(* CODESYS project tcunit.library
   Company: www.tcunit.org
   DefaultNamespace: TcUnit
   Version: 1.0.0.0
   Placeholder: TcUnit
   Author: Jakob Sagatowski and contributors
   Description: TwinCAT unit testing framework.
      Documentation and examples are available at www.tcunit.org
   Title: TcUnit

Project tree, tasks and I/O mapping:
  libraries: Base Interfaces, * (System); SysFile, * (System); Tc2_Standard, * (Beckhoff Automation GmbH); Tc2_System, * (Beckhoff Automation GmbH); Tc2_Utilities, * (Beckhoff Automation GmbH)
  DUTs/
    data type E_XmlError
    data type ST_ADSLogStringMessage
    data type ST_AssertArrayResult
    data type ST_AssertArrayResultInstances
    data type ST_AssertResult
    data type ST_AssertResultInstances
    data type U_ExpectedOrActual
  GVLs/
    global variables GVL_Param_TcUnit
    global variables GVL_Param_XmlControl
    global variables GVL_TcUnit
  ITFs/
    interface I_AssertMessageFormatter: LogAssertFailure
    interface I_TestResultFormatter: Format
  POUs/
    Functions/
      WRITE_PROTECTED_/
        function WRITE_PROTECTED_BOOL [ST]
        function WRITE_PROTECTED_BYTE [ST]
        function WRITE_PROTECTED_DATE [ST]
        function WRITE_PROTECTED_DATE_AND_TIME [ST]
        function WRITE_PROTECTED_DINT [ST]
        function WRITE_PROTECTED_DWORD [ST]
        function WRITE_PROTECTED_INT [ST]
        function WRITE_PROTECTED_LREAL [ST]
        function WRITE_PROTECTED_REAL [ST]
        function WRITE_PROTECTED_SINT [ST]
        function WRITE_PROTECTED_STRING [ST]
        function WRITE_PROTECTED_TIME [ST]
        function WRITE_PROTECTED_TIME_OF_DAY [ST]
        function WRITE_PROTECTED_UDINT [ST]
        function WRITE_PROTECTED_UINT [ST]
        function WRITE_PROTECTED_USINT [ST]
        function WRITE_PROTECTED_WORD [ST]
      function F_AnyToUnionValue [ST]
      function F_AnyTypeClassToString [ST]
      function F_IsAnyEqualToUnionValue [ST]
      function F_RemoveInstancePathAndProjectNameFromTestInstancePath [ST]
      function IS_TEST_FINISHED [ST]
      function RUN [ST]
      function TEST [ST]
      function TEST_FINISHED [ST]
      function TEST_FINISHED_NAMED [ST]
    function block FB_AdjustAssertFailureMessageToMax252CharLength [ST]
    function block FB_ADSAssertMessageFormatter [ST]: LogAssertFailure
    function block FB_ADSLogStringMessageFifoQueue [ST]: GetLog, GetLogCount, WriteLog
    function block FB_ADSTestResultFormatter [ST]: Format
    function block FB_AnyComparator [ST]
    function block FB_AssertArrayResultStatic [ST]: AddAssertArrayResult, CopyDetectionCountAndResetDetectionCountInThisCycle, CreateAssertResultInstance, GetDetectionCount, GetDetectionCountThisCycle, IncreaseDetectionCountThisCycleByOne, ReportResult
    function block FB_AssertResultStatic [ST]: AddAssertResult, CopyDetectionCountAndResetDetectionCountInThisCycle, CreateAssertResultInstance, GetDetectionCount, GetDetectionCountThisCycle, IncreaseDetectionCountThisCycleByOne, ReportResult
    function block FB_FileControl [ST]: Close, Open, Read, Save
    function block FB_StringBuffer [ST]: Append, BufferSize, Copy, CutOff, Find, FindBack, Length, Set
    function block FB_TcUnitRunner [ST]: AbortRunningTestSuiteTests, RunTestSuiteTests
    function block FB_Test [ST]: GetName, IsFailed, IsFinished, SetFailed, SetFinished, SetName
    function block FB_TestSuite [ST]: AddTest, AddTestNameToInstancePath, AreAllTestsFinished, AssertArray2dEquals_LREAL, AssertArray2dEquals_REAL, AssertArray3dEquals_LREAL, AssertArray3dEquals_REAL, AssertArrayEquals_BOOL, AssertArrayEquals_BYTE, AssertArrayEquals_DINT, AssertArrayEquals_DWORD, AssertArrayEquals_INT, AssertArrayEquals_LINT, AssertArrayEquals_LREAL, AssertArrayEquals_LWORD, AssertArrayEquals_REAL, AssertArrayEquals_SINT, AssertArrayEquals_UDINT, AssertArrayEquals_UINT, AssertArrayEquals_ULINT, AssertArrayEquals_USINT, AssertArrayEquals_WORD, AssertEquals, AssertEquals_BOOL, AssertEquals_BYTE, AssertEquals_DATE, AssertEquals_DATE_AND_TIME, AssertEquals_DINT, AssertEquals_DWORD, AssertEquals_INT, AssertEquals_LINT, AssertEquals_LREAL, AssertEquals_LTIME, AssertEquals_LWORD, AssertEquals_REAL, AssertEquals_SINT, AssertEquals_STRING, AssertEquals_TIME, AssertEquals_TIME_OF_DAY, AssertEquals_UDINT, AssertEquals_UINT, AssertEquals_ULINT, AssertEquals_USINT, AssertEquals_WORD, AssertFalse, AssertTrue, FB_init, FindTestSuiteInstancePath, GetInstancePath, GetNumberOfFailedTests, GetNumberOfSuccessfulTests, GetNumberOfTests, SetTestFailed, SetTestFinished
    function block FB_XmlControl [ST]: ClearBuffer, CloseTag, Length, NewComment, NewParameter, NewTag, NewTagData, NextParameter, NextTag, SetBuffer, ToStartBuffer, WriteDocumentHeader
  Version/
    global variables Global_Version
*)

// DUTs/E_XmlError
{attribute 'qualified_only'}
{attribute 'strict'}
TYPE E_XmlError :
(
    Ok := 0,
    ErrorMaxBufferLen := 1,
    ErrorStringLen := 2,
    Error := 3
) BYTE;
END_TYPE

// DUTs/ST_ADSLogStringMessage
{attribute 'pack_mode' := '1'}
TYPE ST_ADSLogStringMessage :
STRUCT
    MsgFmtStr : Tc2_System.T_MaxString;
    StrArg : Tc2_System.T_MaxString;
END_STRUCT
END_TYPE

// DUTs/ST_AssertArrayResult
TYPE ST_AssertArrayResult :
STRUCT
    ExpectedsSize : UDINT; // Size in bytes of the expecteds-array
    ExpectedsTypeClass : IBaseLibrary.TypeClass; // The data type of the expecteds-array
    ActualsSize : UDINT; // Size in bytes of the actuals-array
    ActualsTypeClass : IBaseLibrary.TypeClass; // The data type of the actuals-array
    Message : Tc2_System.T_MaxString;
    TestInstancePath : Tc2_System.T_MaxString;
END_STRUCT
END_TYPE

// DUTs/ST_AssertArrayResultInstances
TYPE ST_AssertArrayResultInstances :
STRUCT
    AssertArrayResult : ST_AssertArrayResult;
    DetectionCount : UINT; // Number of instances of the "AssertArrayResult"
    DetectionCountThisCycle : UINT; // Number of instance of the "AssertArrayResult" in this specific PLC-cycle
END_STRUCT
END_TYPE

// DUTs/ST_AssertResult
TYPE ST_AssertResult :
STRUCT
    Expected : U_ExpectedOrActual;
    Actual : U_ExpectedOrActual;
    Message : Tc2_System.T_MaxString;
    TestInstancePath : Tc2_System.T_MaxString;
END_STRUCT
END_TYPE

// DUTs/ST_AssertResultInstances
TYPE ST_AssertResultInstances :
STRUCT
    AssertResult : ST_AssertResult;
    DetectionCount : UINT; // Number of instances of the "AssertResult"
    DetectionCountThisCycle : UINT; // Number of instance of the "AssertResult" in this specific PLC-cycle
END_STRUCT
END_TYPE

// DUTs/U_ExpectedOrActual
TYPE U_ExpectedOrActual :
UNION
    boolExpectedOrActual : BOOL;
    bitExpectedOrActual : BIT;
    byteExpectedOrActual : BYTE;
    dwordExpectedOrActual : DWORD;
    lwordExpectedOrActual : LWORD;
    stringExpectedOrActual : Tc2_System.T_MaxString;
    udintExpectedOrActual : UDINT;
    uintExpectedOrActual : UINT;
    usintExpectedOrActual : USINT;
    sintExpectedOrActual : SINT;
    intExpectedOrActual : INT;
    wordExpectedOrActual : WORD;
    dintExpectedOrActual : DINT;
    lintExpectedOrActual : LINT;
    ulintExpectedOrActual : ULINT;
    realExpectedOrActual : REAL;
    lrealExpectedOrActual : LREAL;
    wstringExpectedOrActual : WSTRING;
    timeExpectedOrActual : TIME;
    ltimeExpectedOrActual : LTIME;
    dateExpectedOrActual : DATE;
    dateandtimeExpectedOrActual : DATE_AND_TIME;
    timeofdayExpectedOrActual : TIME_OF_DAY;
END_UNION
END_TYPE

// GVLs/GVL_Param_TcUnit
{attribute 'qualified_only'}
VAR_GLOBAL CONSTANT
    MaxNumberOfTestSuites : UINT := 500;
    MaxNumberOfTestsForEachTestSuite : UINT := 100;
    MaxNumberOfAsserts : UINT := 500;
END_VAR

// GVLs/GVL_Param_XmlControl
{attribute 'qualified_only'}
VAR_GLOBAL CONSTANT
    MaxFileSize : UDINT := 4096;
END_VAR

// GVLs/GVL_TcUnit
{attribute 'no_assign'}
{attribute 'qualified_only'}
VAR_GLOBAL
    TcUnitRunner : FB_TcUnitRunner;

    (* Indication of whether the last instantiated test suite has an assert instance created *)
    TestSuiteIsRegistered : BOOL;

    (* Pointer to current test suite being called *)
    CurrentTestSuiteBeingCalled : POINTER TO FB_TestSuite;

    (* Current name of test being called *)
    CurrentTestNameBeingCalled : Tc2_System.T_MaxString;

    (* This is a flag that indicates that the current test should be ignored, and
       thus that all assertions under it should be ignored as well. A test can be ignored either
       because the user has requested so, or because the test is a duplicate name *)
    IgnoreCurrentTest : BOOL;

    (* The assert function block instance should be 1:1 mapped to
       the test suite instance path. *)
    NumberOfInitializedTestSuites : UINT := 0;
    TestSuiteAddresses : ARRAY[1..GVL_Param_TcUnit.MaxNumberOfTestSuites] OF POINTER TO FB_TestSuite;

    (* Buffered ADS logger for output to the error list *)
    AdsLogger : FB_ADSLogStringMessageFifoQueue;
END_VAR

// Version/Global_Version
{attribute 'TcGenerated'}
{attribute 'no-analysis'}
{attribute 'linkalways'}
// This function has been automatically generated from the project information.
VAR_GLOBAL CONSTANT
	{attribute 'const_non_replaced'}
	stLibVersion_TcUnit : ST_LibVersion := (iMajor := 1, iMinor := 0, iBuild := 0, iRevision := 0, sVersion := '1.0.0.0');
END_VAR

// ITFs/I_AssertMessageFormatter
INTERFACE I_AssertMessageFormatter

METHOD LogAssertFailure
VAR_INPUT
    Expected : Tc2_System.T_MaxString;
    Actual : Tc2_System.T_MaxString;
    Message : Tc2_System.T_MaxString;
    TestInstancePath : Tc2_System.T_MaxString;
END_VAR
END_METHOD

END_INTERFACE

// ITFs/I_TestResultFormatter
INTERFACE I_TestResultFormatter

METHOD Format
VAR_INPUT
    NumberOfTestSuites : UINT; // The total number of test suites
    NumberOfTestCases : UINT; // The total number of test cases (for all test suites)
    NumberOfSuccessfulTestCases : UINT; // The total number of test cases that had all ASSERTS successful
    NumberOfFailedTestCases : UINT; // The total number of test cases that had at least one ASSERT failed
END_VAR
VAR_OUTPUT
    Busy : BOOL;
END_VAR
END_METHOD

END_INTERFACE

// POUs/Functions/TEST
(*
    This function declares a new test (if it has not been already declared in an earlier cycle)
*)
FUNCTION TEST
VAR_INPUT
    TestName : Tc2_System.T_MaxString;
END_VAR
VAR
    CounterTestSuiteAddress : UINT;
    CounterTestName : UINT;
END_VAR

(* Mark this test as the current one being executed *)
GVL_TcUnit.CurrentTestNameBeingCalled := TestName;

(* Check if combination of address for the test suite and test name already exists.
   For every test suite the name of the test case needs to be unique.
   If a test with this name already exists, don't add it to the available tests.
   Otherwise, add it to the available tests *)

FOR CounterTestSuiteAddress := 1 TO GVL_TcUnit.NumberOfInitializedTestSuites BY 1 DO
    (* Look for the test suite by comparing to the one that is currently running *)
    IF GVL_TcUnit.TestSuiteAddresses[CounterTestSuiteAddress] = GVL_TcUnit.CurrentTestSuiteBeingCalled THEN
        GVL_TcUnit.TestSuiteAddresses[CounterTestSuiteAddress]^.AddTest(TestName := TestName);
        RETURN;
    END_IF
END_FOR

END_FUNCTION

// POUs/Functions/WRITE_PROTECTED_/WRITE_PROTECTED_BOOL
FUNCTION WRITE_PROTECTED_BOOL
VAR_INPUT
    Ptr : POINTER TO BOOL;
    Value : BOOL;
END_VAR

Ptr^ := Value;

END_FUNCTION

// POUs/Functions/WRITE_PROTECTED_/WRITE_PROTECTED_BYTE
FUNCTION WRITE_PROTECTED_BYTE
VAR_INPUT
    Ptr : POINTER TO BYTE;
    Value : BYTE;
END_VAR

Ptr^ := Value;

END_FUNCTION

// POUs/Functions/WRITE_PROTECTED_/WRITE_PROTECTED_DATE
FUNCTION WRITE_PROTECTED_DATE
VAR_INPUT
    Ptr : POINTER TO DATE;
    Value : DATE;
END_VAR

Ptr^ := Value;

END_FUNCTION

// POUs/Functions/WRITE_PROTECTED_/WRITE_PROTECTED_DATE_AND_TIME
FUNCTION WRITE_PROTECTED_DATE_AND_TIME
VAR_INPUT
    Ptr : POINTER TO DATE_AND_TIME;
    Value : DATE_AND_TIME;
END_VAR

Ptr^ := Value;

END_FUNCTION

// POUs/Functions/WRITE_PROTECTED_/WRITE_PROTECTED_DINT
FUNCTION WRITE_PROTECTED_DINT
VAR_INPUT
    Ptr : POINTER TO DINT;
    Value : DINT;
END_VAR

Ptr^ := Value;

END_FUNCTION

// POUs/Functions/WRITE_PROTECTED_/WRITE_PROTECTED_DWORD
FUNCTION WRITE_PROTECTED_DWORD
VAR_INPUT
    Ptr : POINTER TO DWORD;
    Value : DWORD;
END_VAR

Ptr^ := Value;

END_FUNCTION

// POUs/Functions/WRITE_PROTECTED_/WRITE_PROTECTED_INT
FUNCTION WRITE_PROTECTED_INT
VAR_INPUT
    Ptr : POINTER TO INT;
    Value : INT;
END_VAR

Ptr^ := Value;

END_FUNCTION

// POUs/Functions/WRITE_PROTECTED_/WRITE_PROTECTED_LREAL
FUNCTION WRITE_PROTECTED_LREAL
VAR_INPUT
    Ptr : POINTER TO LREAL;
    Value : LREAL;
END_VAR

Ptr^ := Value;

END_FUNCTION

// POUs/Functions/WRITE_PROTECTED_/WRITE_PROTECTED_REAL
FUNCTION WRITE_PROTECTED_REAL
VAR_INPUT
    Ptr : POINTER TO REAL;
    Value : REAL;
END_VAR

Ptr^ := Value;

END_FUNCTION

// POUs/Functions/WRITE_PROTECTED_/WRITE_PROTECTED_SINT
FUNCTION WRITE_PROTECTED_SINT
VAR_INPUT
    Ptr : POINTER TO SINT;
    Value : SINT;
END_VAR

Ptr^ := Value;

END_FUNCTION

// POUs/Functions/WRITE_PROTECTED_/WRITE_PROTECTED_STRING
FUNCTION WRITE_PROTECTED_STRING
VAR_INPUT
    Ptr : POINTER TO STRING;
    Value : STRING;
END_VAR

Ptr^ := Value;

END_FUNCTION

// POUs/Functions/WRITE_PROTECTED_/WRITE_PROTECTED_TIME
FUNCTION WRITE_PROTECTED_TIME
VAR_INPUT
    Ptr : POINTER TO TIME;
    Value : TIME;
END_VAR

Ptr^ := Value;

END_FUNCTION

// POUs/Functions/WRITE_PROTECTED_/WRITE_PROTECTED_TIME_OF_DAY
FUNCTION WRITE_PROTECTED_TIME_OF_DAY
VAR_INPUT
    Ptr : POINTER TO TIME_OF_DAY;
    Value : TIME_OF_DAY;
END_VAR

Ptr^ := Value;

END_FUNCTION

// POUs/Functions/WRITE_PROTECTED_/WRITE_PROTECTED_UDINT
FUNCTION WRITE_PROTECTED_UDINT
VAR_INPUT
    Ptr : POINTER TO UDINT;
    Value : UDINT;
END_VAR

Ptr^ := Value;

END_FUNCTION

// POUs/Functions/WRITE_PROTECTED_/WRITE_PROTECTED_UINT
FUNCTION WRITE_PROTECTED_UINT
VAR_INPUT
    Ptr : POINTER TO UINT;
    Value : UINT;
END_VAR

Ptr^ := Value;

END_FUNCTION

// POUs/Functions/WRITE_PROTECTED_/WRITE_PROTECTED_USINT
FUNCTION WRITE_PROTECTED_USINT
VAR_INPUT
    Ptr : POINTER TO USINT;
    Value : USINT;
END_VAR

Ptr^ := Value;

END_FUNCTION

// POUs/Functions/WRITE_PROTECTED_/WRITE_PROTECTED_WORD
FUNCTION WRITE_PROTECTED_WORD
VAR_INPUT
    Ptr : POINTER TO WORD;
    Value : WORD;
END_VAR

Ptr^ := Value;

END_FUNCTION

// POUs/Functions/F_AnyToUnionValue
FUNCTION F_AnyToUnionValue : U_ExpectedOrActual
VAR_INPUT
    AnyValue : ANY;
END_VAR

CASE UDINT_TO_INT(AnyValue.TypeClass) OF
    IBaseLibrary.TypeClass.TYPE_BOOL :
        Tc2_System.MEMCPY(destaddr := ADR(F_AnyToUnionValue.boolExpectedOrActual),
                          srcAddr := AnyValue.pValue,
                          n := DINT_TO_UDINT(AnyValue.diSize));

    IBaseLibrary.TypeClass.TYPE_BIT :
        {warning disable C0355}
        Tc2_System.MEMCPY(destaddr := ADR(F_AnyToUnionValue.bitExpectedOrActual),
                          srcAddr := AnyValue.pValue,
                          n := DINT_TO_UDINT(AnyValue.diSize));
        {warning enable C0355}

    IBaseLibrary.TypeClass.TYPE_BYTE :
        Tc2_System.MEMCPY(destaddr := ADR(F_AnyToUnionValue.byteExpectedOrActual),
                          srcAddr := AnyValue.pValue,
                          n := DINT_TO_UDINT(AnyValue.diSize));

    IBaseLibrary.TypeClass.TYPE_WORD :
        Tc2_System.MEMCPY(destaddr := ADR(F_AnyToUnionValue.wordExpectedOrActual),
                          srcAddr := AnyValue.pValue,
                          n := DINT_TO_UDINT(AnyValue.diSize));

    IBaseLibrary.TypeClass.TYPE_DWORD :
        Tc2_System.MEMCPY(destaddr := ADR(F_AnyToUnionValue.dwordExpectedOrActual),
                          srcAddr := AnyValue.pValue,
                          n := DINT_TO_UDINT(AnyValue.diSize));

    IBaseLibrary.TypeClass.TYPE_LWORD :
        Tc2_System.MEMCPY(destaddr := ADR(F_AnyToUnionValue.lwordExpectedOrActual),
                          srcAddr := AnyValue.pValue,
                          n := DINT_TO_UDINT(AnyValue.diSize));

    IBaseLibrary.TypeClass.TYPE_SINT :
        Tc2_System.MEMCPY(destaddr := ADR(F_AnyToUnionValue.sintExpectedOrActual),
                          srcAddr := AnyValue.pValue,
                          n := DINT_TO_UDINT(AnyValue.diSize));

    IBaseLibrary.TypeClass.TYPE_INT :
        Tc2_System.MEMCPY(destaddr := ADR(F_AnyToUnionValue.intExpectedOrActual),
                          srcAddr := AnyValue.pValue,
                          n := DINT_TO_UDINT(AnyValue.diSize));

    IBaseLibrary.TypeClass.TYPE_DINT :
        Tc2_System.MEMCPY(destaddr := ADR(F_AnyToUnionValue.dintExpectedOrActual),
                          srcAddr := AnyValue.pValue,
                          n := DINT_TO_UDINT(AnyValue.diSize));

    IBaseLibrary.TypeClass.TYPE_LINT :
        Tc2_System.MEMCPY(destaddr := ADR(F_AnyToUnionValue.lintExpectedOrActual),
                          srcAddr := AnyValue.pValue,
                          n := DINT_TO_UDINT(AnyValue.diSize));

    IBaseLibrary.TypeClass.TYPE_USINT :
        Tc2_System.MEMCPY(destaddr := ADR(F_AnyToUnionValue.usintExpectedOrActual),
                          srcAddr := AnyValue.pValue,
                          n := DINT_TO_UDINT(AnyValue.diSize));

    IBaseLibrary.TypeClass.TYPE_UINT :
        Tc2_System.MEMCPY(destaddr := ADR(F_AnyToUnionValue.uintExpectedOrActual),
                          srcAddr := AnyValue.pValue,
                          n := DINT_TO_UDINT(AnyValue.diSize));

    IBaseLibrary.TypeClass.TYPE_UDINT :
        Tc2_System.MEMCPY(destaddr := ADR(F_AnyToUnionValue.udintExpectedOrActual),
                          srcAddr := AnyValue.pValue,
                          n := DINT_TO_UDINT(AnyValue.diSize));

    IBaseLibrary.TypeClass.TYPE_ULINT :
        Tc2_System.MEMCPY(destaddr := ADR(F_AnyToUnionValue.ulintExpectedOrActual),
                          srcAddr := AnyValue.pValue,
                          n := DINT_TO_UDINT(AnyValue.diSize));

    IBaseLibrary.TypeClass.TYPE_REAL :
        Tc2_System.MEMCPY(destaddr := ADR(F_AnyToUnionValue.realExpectedOrActual),
                          srcAddr := AnyValue.pValue,
                          n := DINT_TO_UDINT(AnyValue.diSize));

    IBaseLibrary.TypeClass.TYPE_LREAL :
        Tc2_System.MEMCPY(destaddr := ADR(F_AnyToUnionValue.lrealExpectedOrActual),
                          srcAddr := AnyValue.pValue,
                          n := DINT_TO_UDINT(AnyValue.diSize));

    IBaseLibrary.TypeClass.TYPE_STRING :
        Tc2_System.MEMCPY(destaddr := ADR(F_AnyToUnionValue.stringExpectedOrActual),
                          srcAddr := AnyValue.pValue,
                          n := DINT_TO_UDINT(AnyValue.diSize));

    IBaseLibrary.TypeClass.TYPE_WSTRING :
        Tc2_System.MEMCPY(destaddr := ADR(F_AnyToUnionValue.wstringExpectedOrActual),
                          srcAddr := AnyValue.pValue,
                          n := DINT_TO_UDINT(AnyValue.diSize));

    IBaseLibrary.TypeClass.TYPE_TIME :
        Tc2_System.MEMCPY(destaddr := ADR(F_AnyToUnionValue.timeExpectedOrActual),
                          srcAddr := AnyValue.pValue,
                          n := DINT_TO_UDINT(AnyValue.diSize));

    IBaseLibrary.TypeClass.TYPE_DATE :
        Tc2_System.MEMCPY(destaddr := ADR(F_AnyToUnionValue.dateExpectedOrActual),
                          srcAddr := AnyValue.pValue,
                          n := DINT_TO_UDINT(AnyValue.diSize));

    IBaseLibrary.TypeClass.TYPE_DATEANDTIME :
        Tc2_System.MEMCPY(destaddr := ADR(F_AnyToUnionValue.dateandtimeExpectedOrActual),
                          srcAddr := AnyValue.pValue,
                          n := DINT_TO_UDINT(AnyValue.diSize));

    IBaseLibrary.TypeClass.TYPE_TIMEOFDAY :
        Tc2_System.MEMCPY(destaddr := ADR(F_AnyToUnionValue.timeofdayExpectedOrActual),
                          srcAddr := AnyValue.pValue,
                          n := DINT_TO_UDINT(AnyValue.diSize));

    IBaseLibrary.TypeClass.TYPE_POINTER :
        (* None *)

    IBaseLibrary.TypeClass.TYPE_REFERENCE :
        (* None *)

    IBaseLibrary.TypeClass.TYPE_SUBRANGE :
        (* None *)

    IBaseLibrary.TypeClass.TYPE_ENUM :
        (* None *)

    IBaseLibrary.TypeClass.TYPE_ARRAY :
        (* None *)

    IBaseLibrary.TypeClass.TYPE_PARAMS :
        (* None *)

    IBaseLibrary.TypeClass.TYPE_USERDEF :
        (* None *)

    IBaseLibrary.TypeClass.TYPE_NONE :
        (* None *)

    IBaseLibrary.TypeClass.TYPE_ANY :
        (* None *)

    IBaseLibrary.TypeClass.TYPE_ANYBIT :
        (* None *)

    IBaseLibrary.TypeClass.TYPE_ANYDATE :
        (* None *)

    IBaseLibrary.TypeClass.TYPE_ANYINT :
        (* None *)

    IBaseLibrary.TypeClass.TYPE_ANYNUM :
        (* None *)

    IBaseLibrary.TypeClass.TYPE_ANYREAL :
        (* None *)

    IBaseLibrary.TypeClass.TYPE_LAZY :
        (* None *)

    IBaseLibrary.TypeClass.TYPE_LTIME :
        Tc2_System.MEMCPY(destaddr := ADR(F_AnyToUnionValue.ltimeExpectedOrActual),
                          srcAddr := AnyValue.pValue,
                          n := DINT_TO_UDINT(AnyValue.diSize));

    IBaseLibrary.TypeClass.TYPE_BITCONST :
        (* None *)

    IBaseLibrary.TypeClass.TYPE_INTERFACE :
        (* None *)

    ELSE
        (* None *)
END_CASE

END_FUNCTION

// POUs/Functions/F_AnyTypeClassToString
(*
    This function takes the type-class of a ANY-variable and returns the STRING representation of it.
*)
FUNCTION F_AnyTypeClassToString : STRING
VAR_INPUT
    AnyTypeClass : __System.TYPE_CLASS;
END_VAR

CASE UDINT_TO_INT(AnyTypeClass) OF
    IBaseLibrary.TypeClass.TYPE_BOOL :
        F_AnyTypeClassToString := 'BOOL';
    IBaseLibrary.TypeClass.TYPE_BIT :
        F_AnyTypeClassToString := 'BIT';
    IBaseLibrary.TypeClass.TYPE_BYTE :
        F_AnyTypeClassToString := 'BYTE';
    IBaseLibrary.TypeClass.TYPE_WORD :
        F_AnyTypeClassToString := 'WORD';
    IBaseLibrary.TypeClass.TYPE_DWORD :
        F_AnyTypeClassToString := 'DWORD';
    IBaseLibrary.TypeClass.TYPE_LWORD :
        F_AnyTypeClassToString := 'LWORD';
    IBaseLibrary.TypeClass.TYPE_SINT :
        F_AnyTypeClassToString := 'SINT';
    IBaseLibrary.TypeClass.TYPE_INT :
        F_AnyTypeClassToString := 'INT';
    IBaseLibrary.TypeClass.TYPE_DINT :
        F_AnyTypeClassToString := 'DINT';
    IBaseLibrary.TypeClass.TYPE_LINT :
        F_AnyTypeClassToString := 'LINT';
    IBaseLibrary.TypeClass.TYPE_USINT :
        F_AnyTypeClassToString := 'USINT';
    IBaseLibrary.TypeClass.TYPE_UINT :
        F_AnyTypeClassToString := 'UINT';
    IBaseLibrary.TypeClass.TYPE_UDINT :
        F_AnyTypeClassToString := 'UDINT';
    IBaseLibrary.TypeClass.TYPE_ULINT :
        F_AnyTypeClassToString := 'ULINT';
    IBaseLibrary.TypeClass.TYPE_REAL :
        F_AnyTypeClassToString := 'REAL';
    IBaseLibrary.TypeClass.TYPE_LREAL :
        F_AnyTypeClassToString := 'LREAL';
    IBaseLibrary.TypeClass.TYPE_STRING :
        F_AnyTypeClassToString := 'STRING';
    IBaseLibrary.TypeClass.TYPE_WSTRING :
        F_AnyTypeClassToString := 'WSTRING';
    IBaseLibrary.TypeClass.TYPE_TIME :
        F_AnyTypeClassToString := 'TIME';
    IBaseLibrary.TypeClass.TYPE_DATE :
        F_AnyTypeClassToString := 'DATE';
    IBaseLibrary.TypeClass.TYPE_DATEANDTIME :
        F_AnyTypeClassToString := 'DATEANDTIME';
    IBaseLibrary.TypeClass.TYPE_TIMEOFDAY :
        F_AnyTypeClassToString := 'TIMEOFDAY';
    IBaseLibrary.TypeClass.TYPE_POINTER :
        F_AnyTypeClassToString := 'POINTER';
    IBaseLibrary.TypeClass.TYPE_REFERENCE :
        F_AnyTypeClassToString := 'REFERENCE';
    IBaseLibrary.TypeClass.TYPE_SUBRANGE :
        F_AnyTypeClassToString := 'SUBRANGE';
    IBaseLibrary.TypeClass.TYPE_ENUM :
        F_AnyTypeClassToString := 'ENUM';
    IBaseLibrary.TypeClass.TYPE_ARRAY :
        F_AnyTypeClassToString := 'ARRAY';
    IBaseLibrary.TypeClass.TYPE_PARAMS :
        F_AnyTypeClassToString := 'PARAMS';
    IBaseLibrary.TypeClass.TYPE_USERDEF :
        F_AnyTypeClassToString := 'USERDEF';
    IBaseLibrary.TypeClass.TYPE_NONE :
        F_AnyTypeClassToString := 'NONE';
    IBaseLibrary.TypeClass.TYPE_ANY :
        F_AnyTypeClassToString := 'ANY';
    IBaseLibrary.TypeClass.TYPE_ANYBIT :
        F_AnyTypeClassToString := 'ANYBIT';
    IBaseLibrary.TypeClass.TYPE_ANYDATE :
        F_AnyTypeClassToString := 'ANYDATE';
    IBaseLibrary.TypeClass.TYPE_ANYINT :
        F_AnyTypeClassToString := 'ANYINT';
    IBaseLibrary.TypeClass.TYPE_ANYNUM :
        F_AnyTypeClassToString := 'ANYNUM';
    IBaseLibrary.TypeClass.TYPE_ANYREAL :
        F_AnyTypeClassToString := 'ANYREAL';
    IBaseLibrary.TypeClass.TYPE_LAZY :
        F_AnyTypeClassToString := 'LAZY';
    IBaseLibrary.TypeClass.TYPE_LTIME :
        F_AnyTypeClassToString := 'LTIME';
    IBaseLibrary.TypeClass.TYPE_BITCONST :
        F_AnyTypeClassToString := 'BITCONST';
    IBaseLibrary.TypeClass.TYPE_INTERFACE :
        F_AnyTypeClassToString := 'INTERFACE';
    ELSE
        F_AnyTypeClassToString := 'UNKNOWN';
END_CASE

END_FUNCTION

// POUs/Functions/F_IsAnyEqualToUnionValue
FUNCTION F_IsAnyEqualToUnionValue : BOOL
VAR_INPUT
    uExpectedOrActual : U_ExpectedOrActual;
    ExpectedOrActual : ANY;
END_VAR
VAR
    AnyExpectedOrActual : U_ExpectedOrActual;
END_VAR

AnyExpectedOrActual := F_AnyToUnionValue(ExpectedOrActual);

CASE UDINT_TO_INT(ExpectedOrActual.TypeClass) OF

    IBaseLibrary.TypeClass.TYPE_BOOL :
        F_IsAnyEqualToUnionValue := uExpectedOrActual.boolExpectedOrActual = AnyExpectedOrActual.boolExpectedOrActual;

    IBaseLibrary.TypeClass.TYPE_BIT :
        F_IsAnyEqualToUnionValue := uExpectedOrActual.bitExpectedOrActual = AnyExpectedOrActual.bitExpectedOrActual;

    IBaseLibrary.TypeClass.TYPE_BYTE :
        F_IsAnyEqualToUnionValue := uExpectedOrActual.byteExpectedOrActual = AnyExpectedOrActual.byteExpectedOrActual;

    IBaseLibrary.TypeClass.TYPE_WORD :
        F_IsAnyEqualToUnionValue := uExpectedOrActual.wordExpectedOrActual = AnyExpectedOrActual.wordExpectedOrActual;

    IBaseLibrary.TypeClass.TYPE_DWORD :
        F_IsAnyEqualToUnionValue := uExpectedOrActual.dwordExpectedOrActual = AnyExpectedOrActual.dwordExpectedOrActual;

    IBaseLibrary.TypeClass.TYPE_LWORD :
        F_IsAnyEqualToUnionValue := uExpectedOrActual.lwordExpectedOrActual = AnyExpectedOrActual.lwordExpectedOrActual;

    IBaseLibrary.TypeClass.TYPE_SINT :
        F_IsAnyEqualToUnionValue := uExpectedOrActual.sintExpectedOrActual = AnyExpectedOrActual.sintExpectedOrActual;

    IBaseLibrary.TypeClass.TYPE_INT :
        F_IsAnyEqualToUnionValue := uExpectedOrActual.intExpectedOrActual = AnyExpectedOrActual.intExpectedOrActual;

    IBaseLibrary.TypeClass.TYPE_DINT :
        F_IsAnyEqualToUnionValue := uExpectedOrActual.dintExpectedOrActual = AnyExpectedOrActual.dintExpectedOrActual;

    IBaseLibrary.TypeClass.TYPE_LINT :
        F_IsAnyEqualToUnionValue := uExpectedOrActual.lintExpectedOrActual = AnyExpectedOrActual.lintExpectedOrActual;

    IBaseLibrary.TypeClass.TYPE_USINT :
        F_IsAnyEqualToUnionValue := uExpectedOrActual.usintExpectedOrActual = AnyExpectedOrActual.usintExpectedOrActual;

    IBaseLibrary.TypeClass.TYPE_UINT :
        F_IsAnyEqualToUnionValue := uExpectedOrActual.uintExpectedOrActual = AnyExpectedOrActual.uintExpectedOrActual;

    IBaseLibrary.TypeClass.TYPE_UDINT :
        F_IsAnyEqualToUnionValue := uExpectedOrActual.udintExpectedOrActual = AnyExpectedOrActual.udintExpectedOrActual;

    IBaseLibrary.TypeClass.TYPE_ULINT :
        F_IsAnyEqualToUnionValue := uExpectedOrActual.ulintExpectedOrActual = AnyExpectedOrActual.ulintExpectedOrActual;

    IBaseLibrary.TypeClass.TYPE_REAL :
        F_IsAnyEqualToUnionValue := uExpectedOrActual.realExpectedOrActual = AnyExpectedOrActual.realExpectedOrActual;

    IBaseLibrary.TypeClass.TYPE_LREAL :
        F_IsAnyEqualToUnionValue := uExpectedOrActual.lrealExpectedOrActual = AnyExpectedOrActual.lrealExpectedOrActual;

    IBaseLibrary.TypeClass.TYPE_STRING :
        F_IsAnyEqualToUnionValue := uExpectedOrActual.stringExpectedOrActual = AnyExpectedOrActual.stringExpectedOrActual;

    IBaseLibrary.TypeClass.TYPE_WSTRING :
        F_IsAnyEqualToUnionValue := uExpectedOrActual.wstringExpectedOrActual = AnyExpectedOrActual.wstringExpectedOrActual;

    IBaseLibrary.TypeClass.TYPE_TIME :
        F_IsAnyEqualToUnionValue := uExpectedOrActual.timeExpectedOrActual = AnyExpectedOrActual.timeExpectedOrActual;

    IBaseLibrary.TypeClass.TYPE_DATE :
        F_IsAnyEqualToUnionValue := uExpectedOrActual.dateExpectedOrActual = AnyExpectedOrActual.dateExpectedOrActual;

    IBaseLibrary.TypeClass.TYPE_DATEANDTIME :
        F_IsAnyEqualToUnionValue := uExpectedOrActual.dateandtimeExpectedOrActual = AnyExpectedOrActual.dateandtimeExpectedOrActual;

    IBaseLibrary.TypeClass.TYPE_TIMEOFDAY :
        F_IsAnyEqualToUnionValue := uExpectedOrActual.timeofdayExpectedOrActual = AnyExpectedOrActual.timeofdayExpectedOrActual;

    IBaseLibrary.TypeClass.TYPE_POINTER :
        F_IsAnyEqualToUnionValue := FALSE;

    IBaseLibrary.TypeClass.TYPE_REFERENCE :
        F_IsAnyEqualToUnionValue := FALSE;

    IBaseLibrary.TypeClass.TYPE_SUBRANGE :
        F_IsAnyEqualToUnionValue := FALSE;

    IBaseLibrary.TypeClass.TYPE_ENUM :
        F_IsAnyEqualToUnionValue := FALSE;

    IBaseLibrary.TypeClass.TYPE_ARRAY :
        F_IsAnyEqualToUnionValue := FALSE;

    IBaseLibrary.TypeClass.TYPE_PARAMS :
        F_IsAnyEqualToUnionValue := FALSE;

    IBaseLibrary.TypeClass.TYPE_USERDEF :
        F_IsAnyEqualToUnionValue := FALSE;

    IBaseLibrary.TypeClass.TYPE_NONE :
        F_IsAnyEqualToUnionValue := FALSE;

    IBaseLibrary.TypeClass.TYPE_ANY :
        (* Even though the data input of the ExpectedOrActual is ANY, this CASE-switch will never
           enter this case, but instead the type-class that it is an instance of. So for instance,
           if the ExpectedOrActual is an instance of INT, this case-switch will enter the 
           IBaseLibrary.TypeClass.TYPE_INT case. *)
        F_IsAnyEqualToUnionValue := FALSE;

    IBaseLibrary.TypeClass.TYPE_ANYBIT :
        F_IsAnyEqualToUnionValue := FALSE;

    IBaseLibrary.TypeClass.TYPE_ANYDATE :
        F_IsAnyEqualToUnionValue := FALSE;

    IBaseLibrary.TypeClass.TYPE_ANYINT :
        F_IsAnyEqualToUnionValue := FALSE;

    IBaseLibrary.TypeClass.TYPE_ANYNUM :
        F_IsAnyEqualToUnionValue := FALSE;

    IBaseLibrary.TypeClass.TYPE_ANYREAL :
        F_IsAnyEqualToUnionValue := FALSE;

    IBaseLibrary.TypeClass.TYPE_LAZY :
        F_IsAnyEqualToUnionValue := FALSE;

    IBaseLibrary.TypeClass.TYPE_LTIME :
        F_IsAnyEqualToUnionValue := uExpectedOrActual.ltimeExpectedOrActual = AnyExpectedOrActual.ltimeExpectedOrActual;

    IBaseLibrary.TypeClass.TYPE_BITCONST :
        F_IsAnyEqualToUnionValue := FALSE;

    IBaseLibrary.TypeClass.TYPE_INTERFACE :
        F_IsAnyEqualToUnionValue := FALSE;

    ELSE
        F_IsAnyEqualToUnionValue := FALSE;
END_CASE

END_FUNCTION

// POUs/Functions/F_RemoveInstancePathAndProjectNameFromTestInstancePath
FUNCTION F_RemoveInstancePathAndProjectNameFromTestInstancePath : Tc2_System.T_MaxString
VAR_INPUT
    TestInstancePath : Tc2_System.T_MaxString;
END_VAR
VAR
    CharacterPositionOfProjectName : INT;
    ProjectNameWithDot : Tc2_System.T_MaxString;
END_VAR

(* Add the '.' character to the project name for search *)
ProjectNameWithDot := Tc2_Standard.CONCAT(STR1 := TwinCAT_SystemInfoVarList._AppInfo.ProjectName, STR2 := '.');

(* Find the character position of the beginning of the first occurence of the project name *)
CharacterPositionOfProjectName := Tc2_Standard.FIND(STR1 := TestInstancePath, STR2 := ProjectNameWithDot);

IF CharacterPositionOfProjectName > 0 THEN
    TestInstancePath := Tc2_Standard.DELETE(STR := TestInstancePath,
                                            LEN := CharacterPositionOfProjectName-1 + Tc2_Standard.LEN(ProjectNameWithDot),
                                            POS := 1);
END_IF

(* Check if the project name happens to be the same as namespace, and in that case, remove that as well *)
CharacterPositionOfProjectName := Tc2_Standard.FIND(STR1 := TestInstancePath,
                                                    STR2 := ProjectNameWithDot);

IF CharacterPositionOfProjectName > 0 THEN
    TestInstancePath := Tc2_Standard.DELETE(STR := TestInstancePath,
                                            LEN := CharacterPositionOfProjectName - 1 + 
                                                Tc2_Standard.LEN(STR := ProjectNameWithDot),
                                            POS := 1);
END_IF

F_RemoveInstancePathAndProjectNameFromTestInstancePath := TestInstancePath;

END_FUNCTION

// POUs/Functions/IS_TEST_FINISHED
(* Check if a certain test in the current suite is finished *)
FUNCTION IS_TEST_FINISHED : BOOL
VAR_INPUT
    TestName : Tc2_System.T_MaxString;
END_VAR
VAR
    Counter : UINT;
    CurrentTest : FB_Test;
END_VAR

IS_TEST_FINISHED := FALSE;

FOR Counter := 1 TO GVL_TcUnit.CurrentTestSuiteBeingCalled^.GetNumberOfTests() BY 1 DO
    CurrentTest := GVL_TcUnit.CurrentTestSuiteBeingCalled^.Tests[Counter];
    IF CurrentTest.TestName = TestName THEN
        IS_TEST_FINISHED := CurrentTest.IsFinished();
        RETURN;
    END_IF
END_FOR

END_FUNCTION

// POUs/FB_Test
(*
    This function block holds all data that defines a test.
*)
FUNCTION_BLOCK FB_Test
VAR
    TestName : Tc2_System.T_MaxString;
    TestIsFailed : BOOL; // Indication of whether this test has at least one failed assert
    TestIsFinished : BOOL;
END_VAR

METHOD PUBLIC GetName : Tc2_System.T_MaxString;
GetName := TestName;
END_METHOD

METHOD PUBLIC IsFailed : BOOL
IsFailed := TestIsFailed;
END_METHOD

METHOD PUBLIC IsFinished : BOOL
IsFinished := TestIsFinished;
END_METHOD

METHOD PUBLIC SetFailed
TestIsFailed := TRUE;
END_METHOD

METHOD SetFinished : BOOL
TestIsFinished := TRUE;
END_METHOD

METHOD PUBLIC SetName
VAR_INPUT
    Name : Tc2_System.T_MaxString;
END_VAR
TestName := Name;
END_METHOD

END_FUNCTION_BLOCK

// POUs/Functions/RUN
(*
    This function runs all test suites that have been initialized.
*)
FUNCTION RUN

GVL_TcUnit.TcUnitRunner.RunTestSuiteTests();

END_FUNCTION

// POUs/Functions/TEST_FINISHED
(* Sets the currently running test as finished *)
FUNCTION TEST_FINISHED : BOOL
VAR
    TestName : Tc2_System.T_MaxString;
    Counter : UINT := 0;
END_VAR

// Grab the currently running test name
TestName := GVL_TcUnit.CurrentTestNameBeingCalled;

TEST_FINISHED := FALSE;
// Find the test suite and set the test in that test suite as finished
FOR Counter := 1 TO GVL_TcUnit.NumberOfInitializedTestSuites BY 1 DO
    IF GVL_TcUnit.TestSuiteAddresses[Counter] = GVL_TcUnit.CurrentTestSuiteBeingCalled THEN
        GVL_TcUnit.TestSuiteAddresses[Counter]^.SetTestFinished(TestName := GVL_TcUnit.CurrentTestNameBeingCalled);
        TEST_FINISHED := TRUE;
        RETURN;
    END_IF
END_FOR

END_FUNCTION

// POUs/Functions/TEST_FINISHED_NAMED
(* Sets a test defined by TestName as finished. Note that the TestName-input must match
   a TestName that has been previously defined in this test suite. *)
FUNCTION TEST_FINISHED_NAMED
VAR_INPUT
    TestName : Tc2_System.T_MaxString;
END_VAR
VAR
    Counter : UINT := 0;
END_VAR
VAR_STAT
    FailedLookupCounter : UINT := 0;
    AlreadyPrintedFinalWarning : BOOL := FALSE;
END_VAR
VAR CONSTANT
    MaxNumberOfNonExistentTestNamesFailedLookups : UINT := 3;
END_VAR

// Find the test suite and set the test in that test suite as finished
FOR Counter := 1 TO GVL_TcUnit.NumberOfInitializedTestSuites BY 1 DO
    IF GVL_TcUnit.TestSuiteAddresses[Counter] = GVL_TcUnit.CurrentTestSuiteBeingCalled THEN
        IF NOT GVL_TcUnit.TestSuiteAddresses[Counter]^.SetTestFinished(TestName := TestName) AND
            FailedLookupCounter < MaxNumberOfNonExistentTestNamesFailedLookups THEN
            GVL_TcUnit.AdsLogger.WriteLog(MsgFmtStr := 'Failed to find test $'%s$'',
                                          StrArg := TestName);
            FailedLookupCounter := FailedLookupCounter + 1;
            (* Abort TcUnit *)
            GVL_TcUnit.TcUnitRunner.AbortRunningTestSuiteTests();
        ELSIF NOT AlreadyPrintedFinalWarning THEN
            GVL_TcUnit.AdsLogger.WriteLog(MsgFmtStr := 'Excess failed attempts to mark test finished, failed. Further warnings will be suppressed',
                                          StrArg := TestName);
            AlreadyPrintedFinalWarning := TRUE;
        END_IF
        RETURN;
    END_IF
END_FOR

END_FUNCTION

// POUs/FB_AdjustAssertFailureMessageToMax252CharLength
(*
    This function block is responsible for making sure that the asserted test instance path and test message are not
    loo long. The total printed message can not be more than 252 characters long.
*)
FUNCTION_BLOCK FB_AdjustAssertFailureMessageToMax252CharLength
VAR_INPUT
    MsgFmtString : Tc2_System.T_MaxString; // Test instance path
    StringArg : Tc2_System.T_MaxString; // Test message
END_VAR
VAR_OUTPUT
    MsgFmtStringProcessed : Tc2_System.T_MaxString;
    StringArgProcessed : Tc2_System.T_MaxString;
END_VAR
VAR
    MsgFmtStringTemp : Tc2_System.T_MaxString;
    TestNameTooLong : STRING := '...TestName too long';
    TestMsgTooLong : STRING := '...TestMsg too long';
END_VAR
VAR CONSTANT
    MSG_FMT_STRING_MAX_NUMBER_OF_CHARACTERS : INT := 252; // This is actually 253, but if StrArg-argument is used (which it is in TcUnit) it is 252.
END_VAR

// Check if any of the two strings are too long (or the combination of them)

// All OK
IF (Tc2_Standard.LEN(STR := MsgFmtString) + LEN(STR := StringArg)) <= MSG_FMT_STRING_MAX_NUMBER_OF_CHARACTERS THEN
    MsgFmtStringProcessed := MsgFmtString;
    StringArgProcessed := StringArg;
// If test instance path is longer than 252 chars, shorten it down to 252 characters and additionally with the length of the '...TestName too long'. Add the text '...TestName too long' to the test instance path. Leave no characters for the message.
ELSIF Tc2_Standard.LEN(STR := MsgFmtString) > MSG_FMT_STRING_MAX_NUMBER_OF_CHARACTERS THEN
    MsgFmtStringTemp := Tc2_Standard.LEFT(STR := MsgFmtString, SIZE := (MSG_FMT_STRING_MAX_NUMBER_OF_CHARACTERS - Tc2_Standard.LEN(STR := TestNameTooLong)));
    MsgFmtStringProcessed := Tc2_Standard.CONCAT(STR1 := MsgFmtStringTemp, STR2 := TestNameTooLong);
    StringArgProcessed := '';
// If test message is too long (so we cant fit the text "...TestMsg too long") to the end of it, shorten it so that we can.
ELSIF (MSG_FMT_STRING_MAX_NUMBER_OF_CHARACTERS - Tc2_Standard.LEN(STR := TestMsgTooLong)) >= Tc2_Standard.LEN(STR := MsgFmtString) THEN
    MsgFmtStringProcessed := MsgFmtString;
    StringArgProcessed := Tc2_Standard.LEFT(STR := StringArg,
                                            SIZE := (MSG_FMT_STRING_MAX_NUMBER_OF_CHARACTERS - Tc2_Standard.LEN(STR := TestMsgTooLong) - Tc2_Standard.LEN(STR := MsgFmtStringProcessed)));
    StringArgProcessed := Tc2_Standard.CONCAT(STR1 := StringArgProcessed, STR2 := TestMsgTooLong);
// If test instance path is too long (length is between 232 and 252 characters long), shorten it and add the text '...TestName too long'. Leave no characters for the message
ELSE
    MsgFmtStringTemp := Tc2_Standard.LEFT(STR := MsgFmtString, SIZE := (MSG_FMT_STRING_MAX_NUMBER_OF_CHARACTERS - Tc2_Standard.LEN(STR := TestNameTooLong)));
    MsgFmtStringProcessed := Tc2_Standard.CONCAT(STR1 := MsgFmtStringTemp, STR2 := TestNameTooLong);
    StringArgProcessed := '';
END_IF

END_FUNCTION_BLOCK

// POUs/FB_ADSAssertMessageFormatter
(*
    This function block is responsible for printing the results of the assertions using the built-in
    ADSLOGSTR functionality provided by the Tc2_System library. This sends the result using ADS, which
    is consumed by the error list of Visual Studio.
*)
FUNCTION_BLOCK FB_ADSAssertMessageFormatter IMPLEMENTS I_AssertMessageFormatter

METHOD LogAssertFailure
VAR_INPUT
    Expected : Tc2_System.T_MaxString;
    Actual : Tc2_System.T_MaxString;
    Message : Tc2_System.T_MaxString;
    TestInstancePath : Tc2_System.T_MaxString;
END_VAR
VAR
    AdjustAssertFailureMessageToMax252CharLength : FB_AdjustAssertFailureMessageToMax252CharLength;
    TestInstancePathCleaned : Tc2_System.T_MaxString;
    TestInstancePathFinal : Tc2_System.T_MaxString;
    ReturnValue : DINT;
    TestInstancePathProcessed : Tc2_System.T_MaxString;
    MessageProcessed : Tc2_System.T_MaxString;
END_VAR
TestInstancePathCleaned := F_RemoveInstancePathAndProjectNameFromTestInstancePath(TestInstancePath);
TestInstancePathFinal := Tc2_Standard.CONCAT(STR1 := 'FAILED TEST $'', STR2 := TestInstancePathCleaned);
TestInstancePathFinal := Tc2_Standard.CONCAT(STR1 := TestInstancePathFinal, STR2 := '$'');

IF Tc2_Standard.LEN(STR := Expected) > 0 THEN
    TestInstancePathFinal := Tc2_Standard.CONCAT(STR1 := TestInstancePathFinal, STR2 := ', EXP: ');
    TestInstancePathFinal := Tc2_Standard.CONCAT(STR1 := TestInstancePathFinal, STR2 := Expected);
END_IF
IF Tc2_Standard.LEN(STR := Actual) > 0 THEN
    TestInstancePathFinal := Tc2_Standard.CONCAT(STR1 := TestInstancePathFinal, STR2 := ', ACT: ');
    TestInstancePathFinal := Tc2_Standard.CONCAT(STR1 := TestInstancePathFinal, STR2 := Actual);
END_IF
IF Tc2_Standard.LEN(STR := Message) > 0 THEN
    TestInstancePathFinal := Tc2_Standard.CONCAT(STR1 := TestInstancePathFinal, STR2 := ', MSG: %s ');
END_IF

AdjustAssertFailureMessageToMax252CharLength(MsgFmtString := TestInstancePathFinal,
                                             StringArg := Message,
                                             MsgFmtStringProcessed => TestInstancePathProcessed,
                                             StringArgProcessed => MessageProcessed);

GVL_TcUnit.AdsLogger.WriteLog(MsgFmtStr := TestInstancePathProcessed,
                              StrArg := MessageProcessed);
(*
ReturnValue := Tc2_System.ADSLOGSTR(msgCtrlMask := Tc2_System.ADSLOG_MSGTYPE_ERROR,
                                    msgFmtStr := TestInstancePathProcessed,
                                    strArg := MessageProcessed); *)
END_METHOD

END_FUNCTION_BLOCK

// POUs/FB_ADSLogStringMessageFifoQueue
(* This function block is responsible for making sure that the ADSLOGSTR-messages to the ADS-router are transmitted
   cyclically and not in a burst. The reason this is necessary is because that if too many messages are sent at the
   same time some get lost and are never printed to the error list output
*)
FUNCTION_BLOCK FB_ADSLogStringMessageFifoQueue
VAR
    ArrayBuffer : ARRAY[0..((RING_BUFFER_SIZE * (SIZEOF(ST_ADSLogStringMessage) + MEM_RING_BUFFER_INTERNAL_USE_PER_DATA_RECORD)) - 1)] OF BYTE;
    MemRingBuffer : Tc2_Utilities.FB_MemRingBuffer;
    TimerBetweenMessages : Tc2_Standard.TON := (IN := TRUE, PT := TIME_BETWEEN_MESSAGES);
END_VAR
VAR CONSTANT
    RING_BUFFER_SIZE : UINT := 1000;
    MEM_RING_BUFFER_INTERNAL_USE_PER_DATA_RECORD : USINT := 4;
    TIME_BETWEEN_MESSAGES : TIME := T#50MS;
END_VAR
VAR_TEMP
    MessageToBeSent : ST_ADSLogStringMessage;
    ErrorGet : BOOL;
    ReturnValue : DINT;
END_VAR

TimerBetweenMessages();
IF GetLogCount() > 0 THEN
    // Timer has elapsed, print message
    IF TimerBetweenMessages.Q THEN
        GetLog(AdsLogStringMessage => MessageToBeSent,
               Error => ErrorGet);
        IF NOT ErrorGet THEN
            ReturnValue := Tc2_System.ADSLOGSTR(msgCtrlMask := Tc2_System.ADSLOG_MSGTYPE_ERROR,
                                                msgFmtStr := MessageToBeSent.MsgFmtStr,
                                                strArg := MessageToBeSent.StrArg);
        END_IF
        TimerBetweenMessages(IN := FALSE); // Reset timer
        TimerBetweenMessages.IN := TRUE;
    END_IF
END_IF

(* Reads and removes the oldest message *)
METHOD PRIVATE GetLog
VAR_OUTPUT
    AdsLogStringMessage : ST_ADSLogStringMessage;
    Error : BOOL; // Buffer empty
END_VAR
MemRingBuffer.A_RemoveHead(pRead := ADR(AdsLogStringMessage),
                           cbRead := SIZEOF(ST_ADSLogStringMessage),
                           pBuffer := ADR(ArrayBuffer),
                           cbBuffer := SIZEOF(ArrayBuffer));
Error := NOT MemRingBuffer.bOk;
END_METHOD

METHOD PRIVATE GetLogCount : UDINT
GetLogCount := MemRingBuffer.nCount;
END_METHOD

(* Writes a new data set into the ring buffer *)
METHOD PUBLIC WriteLog
VAR_INPUT
    MsgFmtStr : Tc2_System.T_MaxString;
    StrArg : Tc2_System.T_MaxString;
END_VAR
VAR_OUTPUT
    Error : BOOL; // Buffer overflow
END_VAR
VAR
    AdsLogStringMessage : ST_ADSLogStringMessage;
END_VAR
AdsLogStringMessage.MsgFmtStr := MsgFmtStr;
AdsLogStringMessage.StrArg := StrArg;

MemRingBuffer.A_AddTail(pWrite := ADR(AdsLogStringMessage),
                        cbWrite := SIZEOF(ST_ADSLogStringMessage),
                        pBuffer := ADR(ArrayBuffer),
                        cbBuffer := SIZEOF(ArrayBuffer));

Error := NOT MemRingBuffer.bOk;
END_METHOD

END_FUNCTION_BLOCK

// POUs/FB_ADSTestResultFormatter
(*
    This function block reports the results from the tests using the built-in ADSLOGSTR functionality
    provided by the Tc2_System library. This sends the result using ADS, which is consumed by the error list
    of Visual Studio.
*)
FUNCTION_BLOCK FB_ADSTestResultFormatter IMPLEMENTS I_TestResultFormatter
VAR
    (* Although we can print a message no #1 prior to message no #2, the message #2 can still be displayed before
       message #1, most likely because of some delay of the ADS data. To workaround this, we add a small delay between
       transmission of the ADS messages. *)
    ADSDelayTimer : Tc2_Standard.TON := (PT := T#300MS);
    LastPrintState : USINT := 0;
    PrintState : USINT := 0;
END_VAR

METHOD Format
VAR_INPUT
    (* The total number of test suites *)
    NumberOfTestSuites : UINT;
    (* The total number of test cases (for all test function blocks) *)
    NumberOfTestCases : UINT;
    (* The total number of test cases that had all ASSERTS successful *)
    NumberOfSuccessfulTestCases : UINT;
    (* The total number of test cases that had at least one ASSERT failed *)
    NumberOfFailedTestCases : UINT;
END_VAR
VAR_OUTPUT
    Busy : BOOL;
END_VAR
VAR
    ErrorCode : DINT;
END_VAR
CASE PrintState OF
    0 :
        LastPrintState := PrintState;
        PrintState := 100;
        Busy := TRUE;
    1 :
        GVL_TcUnit.AdsLogger.WriteLog(MsgFmtStr := '%s',
                                      StrArg := '| ==========TESTS FINISHED RUNNING==========');
        LastPrintState := PrintState;
        PrintState := 100;
        Busy := TRUE;
    2 :
        GVL_TcUnit.AdsLogger.WriteLog(MsgFmtStr := '| Test suites: %s',
                                      StrArg := UINT_TO_STRING(NumberOfTestSuites));
        LastPrintState := PrintState;
        PrintState := 100;
        Busy := TRUE;
    3 :
        GVL_TcUnit.AdsLogger.WriteLog(MsgFmtStr := '| Tests: %s',
                                      StrArg := UINT_TO_STRING(NumberOfTestCases));
        LastPrintState := PrintState;
        PrintState := 100;
        Busy := TRUE;
    4 :
        GVL_TcUnit.AdsLogger.WriteLog(MsgFmtStr := '| Successful tests: %s',
                                      StrArg := UINT_TO_STRING(NumberOfSuccessfulTestCases));
        LastPrintState := PrintState;
        PrintState := 100;
        Busy := TRUE;
    5 :
        GVL_TcUnit.AdsLogger.WriteLog(MsgFmtStr := '| Failed tests: %s',
                                      StrArg := UINT_TO_STRING(NumberOfFailedTestCases));
        LastPrintState := PrintState;
        PrintState := 100;
        Busy := TRUE;
    6 :
        GVL_TcUnit.AdsLogger.WriteLog(MsgFmtStr := '%s',
                                      StrArg := '| ======================================');
        LastPrintState := PrintState;
        PrintState := 100;
        Busy := TRUE;
    7 :
        Busy := FALSE;
    100 :
        ADSDelayTimer(IN := TRUE);
        IF ADSDelayTimer.Q THEN
            ADSDelayTimer(IN := FALSE);
            PrintState := LastPrintState + 1;
        END_IF
        Busy := TRUE;
END_CASE
END_METHOD

END_FUNCTION_BLOCK

// POUs/FB_AnyComparator
(*
    This FB compares two instances of any object type and returns whether they
    are the same type, size and value or not. This is necessary for two reasons:
    1. So that we can know exactly what differs between the two input parameters
    2. It's not possible to do a comparison (= or <>) between two instances of ANY.
*)
FUNCTION_BLOCK FB_AnyComparator
VAR_INPUT
    AnyValueOne : ANY;
    AnyValueTwo : ANY;
END_VAR
VAR_OUTPUT
    DataTypesNotEquals : BOOL; // The data type of the two ANY input parameters are not equal
    DataSizeNotEquals : BOOL; // The data size of the two ANY input parameters are not equal
    DataContentNotEquals : BOOL; // The data content of the two ANY input parameters are not equal
END_VAR
VAR
    IteratorCounter : DINT;
END_VAR

(* Reset the outputs *)
DataTypesNotEquals := FALSE;
DataSizeNotEquals := FALSE;
DataContentNotEquals := FALSE;

(* Check whether the type of the inputs differs *)
IF AnyValueOne.TypeClass <> AnyValueTwo.TypeClass THEN
    DataTypesNotEquals := TRUE;
END_IF

(* Check whether the size of the inputs differs *)
IF NOT DataTypesNotEquals THEN
    IF (AnyValueOne.diSize <> AnyValueTwo.diSize) THEN
        DataSizeNotEquals := TRUE;
    END_IF
END_IF

(* Even though the data type and size are equals, the contents may still differ *)
IF NOT DataTypesNotEquals AND NOT DataSizeNotEquals THEN
    // Compare each byte in the ANY-types
    FOR IteratorCounter := 0 TO AnyValueOne.diSize - 1 BY 1 DO
        IF AnyValueOne.pValue[IteratorCounter] <> AnyValueTwo.pValue[IteratorCounter] THEN
            DataContentNotEquals := TRUE;
            EXIT;
        END_IF
    END_FOR
END_IF

END_FUNCTION_BLOCK

// POUs/FB_AssertArrayResultStatic
(*
    This function block is responsible for keeping track of which array-asserts that have been made.
    The reason we need to keep track of these is because if the user does the same assert twice
    (because of running a test suite over several PLC-cycles) we want to know it so we don't print several times
    (if the assert fails). An instance of an array-assert is keyed/identified with the following parameters as key:
    - Array-size (in bytes) of the expecteds
    - Datatype of the expecteds
    - Array-size (in bytes) of the actuals
    - Datatype of the actuals
    - Message (string)
    - Test instance path (string)
*)
FUNCTION_BLOCK FB_AssertArrayResultStatic
VAR
    (* The total number of instances of each of the "AssertArrayResults" *)
    AssertArrayResults : ARRAY[1..GVL_Param_TcUnit.MaxNumberOfAsserts] OF ST_AssertArrayResult;

    (* The total number of unique asserts *)
    TotalArrayAsserts : UINT := 0;

    (* Function block to get the current task cycle *)
    GetCurrentTaskIndex : Tc2_System.GETCURTASKINDEX;

    (* The total number of instances of each of the "AssertArrayResults" *)
    AssertArrayResultInstances : ARRAY[1..GVL_Param_TcUnit.MaxNumberOfAsserts] OF ST_AssertArrayResultInstances;

    (* The last PLC cycle count *)
    CycleCount : UDINT;

    (* Only run first cycle *)
    FirstCycleExecuted : BOOL;
END_VAR

METHOD PRIVATE AddAssertArrayResult
VAR_INPUT
    ExpectedsSize : UDINT;
    ExpectedsTypeClass : IBaseLibrary.TypeClass;
    ActualsSize : UDINT;
    ActualsTypeClass : IBaseLibrary.TypeClass;
    Message : Tc2_System.T_MaxString;
    TestInstancePath : Tc2_System.T_MaxString;
END_VAR
TotalArrayAsserts := TotalArrayAsserts + 1;
AssertArrayResults[TotalArrayAsserts].ExpectedsSize := ExpectedsSize;
AssertArrayResults[TotalArrayAsserts].ExpectedsTypeClass := ExpectedsTypeClass;
AssertArrayResults[TotalArrayAsserts].ActualsSize := ActualsSize;
AssertArrayResults[TotalArrayAsserts].ActualsTypeClass := ActualsTypeClass;
AssertArrayResults[TotalArrayAsserts].Message := Message;
AssertArrayResults[TotalArrayAsserts].TestInstancePath := TestInstancePath;
END_METHOD

METHOD PRIVATE CopyDetectionCountAndResetDetectionCountInThisCycle
VAR
    IteratorCounter : UINT;
END_VAR
FOR IteratorCounter := 1 TO GVL_Param_TcUnit.MaxNumberOfAsserts BY 1 DO
    AssertArrayResultInstances[IteratorCounter].DetectionCount := AssertArrayResultInstances[IteratorCounter].DetectionCountThisCycle;
    AssertArrayResultInstances[IteratorCounter].DetectionCountThisCycle := 0;
END_FOR
END_METHOD

METHOD PRIVATE CreateAssertResultInstance
VAR_INPUT
    ExpectedsSize : UDINT;
    ExpectedsTypeClass : IBaseLibrary.TypeClass;
    ActualsSize : UDINT;
    ActualsTypeClass : IBaseLibrary.TypeClass;
    Message : Tc2_System.T_MaxString;
    TestInstancePath : Tc2_System.T_MaxString;
END_VAR
VAR
    IteratorCounter : UINT;
END_VAR
FOR IteratorCounter := 1 TO GVL_Param_TcUnit.MaxNumberOfAsserts BY 1 DO
    IF AssertArrayResultInstances[IteratorCounter].DetectionCount = 0 AND
        AssertArrayResultInstances[IteratorCounter].DetectionCountThisCycle = 0 THEN // Find first free spot
        AssertArrayResultInstances[IteratorCounter].AssertArrayResult.ExpectedsSize := ExpectedsSize;
        AssertArrayResultInstances[IteratorCounter].AssertArrayResult.ExpectedsTypeClass := ExpectedsTypeClass;
        AssertArrayResultInstances[IteratorCounter].AssertArrayResult.ActualsSize := ActualsSize;
        AssertArrayResultInstances[IteratorCounter].AssertArrayResult.ActualsTypeClass := ActualsTypeClass;
        AssertArrayResultInstances[IteratorCounter].AssertArrayResult.Message := Message;
        AssertArrayResultInstances[IteratorCounter].AssertArrayResult.TestInstancePath := TestInstancePath;
        AssertArrayResultInstances[IteratorCounter].DetectionCountThisCycle := 1;
        EXIT;
    END_IF
END_FOR
END_METHOD

METHOD PRIVATE GetDetectionCount : UINT
VAR_INPUT
    ExpectedsSize : UDINT;
    ExpectedsTypeClass : IBaseLibrary.TypeClass;
    ActualsSize : UDINT;
    ActualsTypeClass : IBaseLibrary.TypeClass;
    Message : Tc2_System.T_MaxString;
    TestInstancePath : Tc2_System.T_MaxString;
END_VAR
VAR
    IteratorCounter : UINT;
END_VAR
FOR IteratorCounter := 1 TO GVL_Param_TcUnit.MaxNumberOfAsserts BY 1 DO
    IF AssertArrayResultInstances[IteratorCounter].AssertArrayResult.ExpectedsSize = ExpectedsSize AND
       AssertArrayResultInstances[IteratorCounter].AssertArrayResult.ExpectedsTypeClass = ExpectedsTypeClass AND
       AssertArrayResultInstances[IteratorCounter].AssertArrayResult.ActualsSize = ActualsSize AND
       AssertArrayResultInstances[IteratorCounter].AssertArrayResult.ActualsTypeClass = ActualsTypeClass AND
        AssertArrayResultInstances[IteratorCounter].AssertArrayResult.Message = Message AND
        AssertArrayResultInstances[IteratorCounter].AssertArrayResult.TestInstancePath = TestInstancePath THEN
        GetDetectionCount := AssertArrayResultInstances[IteratorCounter].DetectionCount;
    END_IF
END_FOR
END_METHOD

METHOD PRIVATE GetDetectionCountThisCycle : UINT
VAR_INPUT
    ExpectedsSize : UDINT;
    ExpectedsTypeClass : IBaseLibrary.TypeClass;
    ActualsSize : UDINT;
    ActualsTypeClass : IBaseLibrary.TypeClass;
    Message : Tc2_System.T_MaxString;
    TestInstancePath : Tc2_System.T_MaxString;
END_VAR
VAR
    IteratorCounter : UINT;
END_VAR
FOR IteratorCounter := 1 TO GVL_Param_TcUnit.MaxNumberOfAsserts BY 1 DO
    IF AssertArrayResultInstances[IteratorCounter].AssertArrayResult.ExpectedsSize = ExpectedsSize AND
       AssertArrayResultInstances[IteratorCounter].AssertArrayResult.ExpectedsTypeClass = ExpectedsTypeClass AND
       AssertArrayResultInstances[IteratorCounter].AssertArrayResult.ActualsSize = ActualsSize AND
       AssertArrayResultInstances[IteratorCounter].AssertArrayResult.ActualsTypeClass = ActualsTypeClass AND
        AssertArrayResultInstances[IteratorCounter].AssertArrayResult.Message = Message AND
        AssertArrayResultInstances[IteratorCounter].AssertArrayResult.TestInstancePath = TestInstancePath THEN

        GetDetectionCountThisCycle := AssertArrayResultInstances[IteratorCounter].DetectionCountThisCycle;
    END_IF
END_FOR
END_METHOD

METHOD PRIVATE IncreaseDetectionCountThisCycleByOne
VAR_INPUT
    ExpectedsSize : UDINT;
    ExpectedsTypeClass : IBaseLibrary.TypeClass;
    ActualsSize : UDINT;
    ActualsTypeClass : IBaseLibrary.TypeClass;
    Message : Tc2_System.T_MaxString;
    TestInstancePath : Tc2_System.T_MaxString;
END_VAR
VAR
    IteratorCounter : UINT;
END_VAR
FOR IteratorCounter := 1 TO GVL_Param_TcUnit.MaxNumberOfAsserts BY 1 DO
    IF AssertArrayResultInstances[IteratorCounter].AssertArrayResult.ExpectedsSize = ExpectedsSize AND
        AssertArrayResultInstances[IteratorCounter].AssertArrayResult.ExpectedsTypeClass = ExpectedsTypeClass AND
        AssertArrayResultInstances[IteratorCounter].AssertArrayResult.ActualsSize = ActualsSize AND
        AssertArrayResultInstances[IteratorCounter].AssertArrayResult.ActualsTypeClass = ActualsTypeClass AND
        AssertArrayResultInstances[IteratorCounter].AssertArrayResult.Message = Message AND
        AssertArrayResultInstances[IteratorCounter].AssertArrayResult.TestInstancePath = TestInstancePath THEN
        AssertArrayResultInstances[IteratorCounter].DetectionCountThisCycle :=
            AssertArrayResultInstances[IteratorCounter].DetectionCountThisCycle + 1;
    END_IF
END_FOR
END_METHOD

(*
    This method is called in every assert and returns whether this particular assert has already been called.
    The reason one would like to know whether this assert has already been reported or not is to not report it several
    times to any logging service. Because a test-suite can consist of several tests, and certain tests can require the
    test to run over several cycles it means that certain asserts could be called several times and thus we need to
    keep track of which asserts we've already reported. The user of the framework should not need to care for any of
    this and he/she should be able to call the asserts in any way they find suitable.

    To know what assert this is we need to check for the total combination of:
    - Test message
    - Test instance path
    - Expecteds size (in bytes)
    - Actuals size (in bytes)
    - Expecteds datatype
    - Actuals datatype
    Theoretically we can have a situation where a test has three different asserts, each and one with the same test
    message/test instance path/actuals size&datatype/expecteds size&datatype but called within the same or different
    cycles. In order for us to handle all situations we need a simple algorithm that works according to:
    - Keep track of how many instances the combination of test message/test instance path/expecteds size&datatype/
      actuals size&datatype we have. So for example, if we have called
      Assert(Exp := [5,4,3], Act := [5,4,3], 'Hello there', 'PRG.InstanceTestSuite.Test')
      two times in one cycle, we have two instances of that combination. This is done according to:
    - Iterate all existing reports.
      - If we have a new PLC-cycle, set the current detection-count to zero.
      - If new report does not match in any of the above fields, create it (together with current PLC-cycle).
        Also store the information that we have one instance of this combination and +1 on the detection-count.
      - If new report matches in all of the above, +1 in the detection-count. If this detection-count is larger than
        the stored detection-count for this combination, create a new report and add +1 to the storage of
        the detection-count.
*)
METHOD PUBLIC ReportResult
VAR_INPUT
    ExpectedsSize : UDINT;
    ExpectedsTypeClass : IBaseLibrary.TypeClass;
    ActualsSize : UDINT;
    ActualsTypeClass : IBaseLibrary.TypeClass;
    Message : Tc2_System.T_MaxString;
    TestInstancePath : Tc2_System.T_MaxString;
END_VAR
VAR_OUTPUT
    AlreadyReported : BOOL := FALSE;
END_VAR
VAR
    LocationIndex : UINT;
    DataTypesNotEquals : BOOL;
    DataSizeNotEquals : BOOL;
    DataContentNotEquals : BOOL;
    CurrentCycleCount : UDINT;
    IteratorCounter : UINT;
    DetectionCountTemp : UINT := 0;
    FoundOne : BOOL;
    AdditionalIdenticalAssert : BOOL;
END_VAR
IF NOT FirstCycleExecuted THEN
    GetCurrentTaskIndex();
    FirstCycleExecuted := TRUE;
END_IF

CurrentCycleCount := TwinCAT_SystemInfoVarList._TaskInfo[GetCurrentTaskIndex.index].CycleCount;
(* Is current cycle the same as the last call to this method?
   If not, reset the detection count *)
IF CurrentCycleCount <> CycleCount THEN
    CopyDetectionCountAndResetDetectionCountInThisCycle();
END_IF

FOR IteratorCounter := 1 TO TotalArrayAsserts BY 1 DO
    IF AssertArrayResultInstances[IteratorCounter].AssertArrayResult.ExpectedsSize = ExpectedsSize AND
        AssertArrayResultInstances[IteratorCounter].AssertArrayResult.ExpectedsTypeClass = ExpectedsTypeClass AND
        AssertArrayResultInstances[IteratorCounter].AssertArrayResult.ActualsSize = ActualsSize AND
        AssertArrayResultInstances[IteratorCounter].AssertArrayResult.ActualsTypeClass = ActualsTypeClass AND
        AssertArrayResultInstances[IteratorCounter].AssertArrayResult.Message = Message AND
        AssertArrayResultInstances[IteratorCounter].AssertArrayResult.TestInstancePath = TestInstancePath THEN
        AssertArrayResultInstances[IteratorCounter].DetectionCountThisCycle :=
            AssertArrayResultInstances[IteratorCounter].DetectionCountThisCycle + 1;
            FoundOne := TRUE;
        IF AssertArrayResultInstances[IteratorCounter].DetectionCountThisCycle >
                AssertArrayResultInstances[IteratorCounter].DetectionCount THEN // This assert is new
                AdditionalIdenticalAssert := TRUE;
        END_IF
        EXIT;
    END_IF
END_FOR

(* If not found anything, create the first *)
IF NOT FoundOne THEN
    (* No existing match found, create a new entry *)
    AddAssertArrayResult(ExpectedsSize, ExpectedsTypeClass, ActualsSize, ActualsTypeClass, Message, TestInstancePath);
    CreateAssertResultInstance(ExpectedsSize, ExpectedsTypeClass, ActualsSize, ActualsTypeClass,
                               Message, TestInstancePath);
(* An additional instance of this assert needs to be created *)
ELSIF AdditionalIdenticalAssert THEN
    AddAssertArrayResult(ExpectedsSize, ExpectedsTypeClass, ActualsSize, ActualsTypeClass, Message, TestInstancePath);
(* In all other cases, this assert has already been reported, we don't need to do anything *)
ELSE
    AlreadyReported := TRUE;
END_IF

(* Update the cycle count *)
CycleCount := TwinCAT_SystemInfoVarList._TaskInfo[GetCurrentTaskIndex.index].CycleCount;
END_METHOD

END_FUNCTION_BLOCK

// POUs/FB_AssertResultStatic
(*
    This function block is responsible for keeping track of which asserts that have been made. The reason we need to
    keep track of these is because if the user does the same assert twice (because of running a test suite over several
    PLC-cycles) we want to know it so we don't print several times (if the assert fails).
    An instance of an assert is keyed/identified with the following parameters as key:
    - Value of expected
    - Value of actual
    - Message (string)
    - Test instance path (string)
*)
FUNCTION_BLOCK FB_AssertResultStatic
VAR
    (* The total number of instances of each of the "AssertResults" *)
    AssertResults : ARRAY[1..GVL_Param_TcUnit.MaxNumberOfAsserts] OF ST_AssertResult;

    (* The total number of unique asserts *)
    TotalAsserts : UINT := 0;

    (* Function block to get the current task cycle *)
    GetCurrentTaskIndex : Tc2_System.GETCURTASKINDEX;

    (* The total number of instances of each of the "AssertResults" *)
    AssertResultInstances : ARRAY[1..GVL_Param_TcUnit.MaxNumberOfAsserts] OF ST_AssertResultInstances;

    (* The last PLC cycle count *)
    CycleCount : UDINT;

    (* Only run first cycle *)
    FirstCycleExecuted : BOOL;
END_VAR

METHOD PRIVATE AddAssertResult
VAR_INPUT
    Expected : ANY;
    Actual : ANY;
    Message : Tc2_System.T_MaxString;
    TestInstancePath : Tc2_System.T_MaxString;
END_VAR
TotalAsserts := TotalAsserts + 1;
AssertResults[TotalAsserts].Expected := F_AnyToUnionValue(AnyValue := Expected);
AssertResults[TotalAsserts].Actual := F_AnyToUnionValue(AnyValue := Actual);
AssertResults[TotalAsserts].Message := Message;
AssertResults[TotalAsserts].TestInstancePath := TestInstancePath;
END_METHOD

METHOD PRIVATE CopyDetectionCountAndResetDetectionCountInThisCycle
VAR
    IteratorCounter : UINT;
END_VAR
FOR IteratorCounter := 1 TO GVL_Param_TcUnit.MaxNumberOfAsserts BY 1 DO
    AssertResultInstances[IteratorCounter].DetectionCount := AssertResultInstances[IteratorCounter].DetectionCountThisCycle;
    AssertResultInstances[IteratorCounter].DetectionCountThisCycle := 0;
END_FOR
END_METHOD

METHOD PRIVATE CreateAssertResultInstance
VAR_INPUT
    Expected : ANY;
    Actual : ANY;
    Message : Tc2_System.T_MaxString;
    TestInstancePath : Tc2_System.T_MaxString;
END_VAR
VAR
    IteratorCounter : UINT;
END_VAR
FOR IteratorCounter := 1 TO GVL_Param_TcUnit.MaxNumberOfAsserts BY 1 DO
    IF AssertResultInstances[IteratorCounter].DetectionCount = 0 AND
        AssertResultInstances[IteratorCounter].DetectionCountThisCycle = 0 THEN // Find first free spot
        AssertResultInstances[IteratorCounter].AssertResult.Expected := F_AnyToUnionValue(AnyValue := Expected);
        AssertResultInstances[IteratorCounter].AssertResult.Actual := F_AnyToUnionValue(AnyValue := Actual);
        AssertResultInstances[IteratorCounter].AssertResult.Message := Message;
        AssertResultInstances[IteratorCounter].AssertResult.TestInstancePath := TestInstancePath;
        AssertResultInstances[IteratorCounter].DetectionCountThisCycle := 1;
        EXIT;
    END_IF
END_FOR
END_METHOD

METHOD PRIVATE GetDetectionCount : UINT
VAR_INPUT
    Expected : ANY;
    Actual : ANY;
    Message : Tc2_System.T_MaxString;
    TestInstancePath : Tc2_System.T_MaxString;
END_VAR
VAR
    IteratorCounter : UINT;
END_VAR
FOR IteratorCounter := 1 TO GVL_Param_TcUnit.MaxNumberOfAsserts BY 1 DO
    IF F_IsAnyEqualToUnionValue(uExpectedOrActual := AssertResultInstances[IteratorCounter].AssertResult.Expected,
                                ExpectedOrActual := Expected) AND 
        F_IsAnyEqualToUnionValue(uExpectedOrActual := AssertResultInstances[IteratorCounter].AssertResult.Actual,
                                 ExpectedOrActual := Actual) AND
        AssertResultInstances[IteratorCounter].AssertResult.Message = Message AND
        AssertResultInstances[IteratorCounter].AssertResult.TestInstancePath = TestInstancePath THEN
        GetDetectionCount := AssertResultInstances[IteratorCounter].DetectionCount;
    END_IF
END_FOR
END_METHOD

METHOD PRIVATE GetDetectionCountThisCycle : UINT
VAR_INPUT
    Expected : ANY;
    Actual : ANY;
    Message : Tc2_System.T_MaxString;
    TestInstancePath : Tc2_System.T_MaxString;
END_VAR
VAR
    IteratorCounter : UINT;
END_VAR
FOR IteratorCounter := 1 TO GVL_Param_TcUnit.MaxNumberOfAsserts BY 1 DO
    IF F_IsAnyEqualToUnionValue(uExpectedOrActual := AssertResultInstances[IteratorCounter].AssertResult.Expected,
                                ExpectedOrActual := Expected) AND 
        F_IsAnyEqualToUnionValue(uExpectedOrActual := AssertResultInstances[IteratorCounter].AssertResult.Actual,
                                 ExpectedOrActual := Actual) AND
        AssertResultInstances[IteratorCounter].AssertResult.Message = Message AND
        AssertResultInstances[IteratorCounter].AssertResult.Message = TestInstancePath THEN
        GetDetectionCountThisCycle := AssertResultInstances[IteratorCounter].DetectionCountThisCycle;
    END_IF
END_FOR
END_METHOD

METHOD PRIVATE IncreaseDetectionCountThisCycleByOne
VAR_INPUT
    Expected : ANY;
    Actual : ANY;
    Message : Tc2_System.T_MaxString;
    TestInstancePath : Tc2_System.T_MaxString;
END_VAR
VAR
    IteratorCounter : UINT;
END_VAR
FOR IteratorCounter := 1 TO GVL_Param_TcUnit.MaxNumberOfAsserts BY 1 DO
    IF F_IsAnyEqualToUnionValue(uExpectedOrActual := AssertResultInstances[IteratorCounter].AssertResult.Expected,
                                ExpectedOrActual := Expected) AND 
        F_IsAnyEqualToUnionValue(uExpectedOrActual := AssertResultInstances[IteratorCounter].AssertResult.Actual,
                                 ExpectedOrActual := Actual) AND
        AssertResultInstances[IteratorCounter].AssertResult.Message = Message AND
        AssertResultInstances[IteratorCounter].AssertResult.TestInstancePath = TestInstancePath THEN
        AssertResultInstances[IteratorCounter].DetectionCountThisCycle :=
            AssertResultInstances[IteratorCounter].DetectionCountThisCycle + 1;
    END_IF
END_FOR
END_METHOD

(*
    This method is called in every assert and returns whether this particular assert has already been called.
    The reason one would like to know whether this assert has already been reported or not is to not report it several
    times to any logging service. Because a test-suite can consist of several tests, and certain tests can require the
    test to run over several cycles it means that certain asserts could be called several times and thus we need to
    keep track of which asserts we've already reported. The user of the framework should not need to care for any of
    this and he/she should be able to call the asserts in any way they find suitable.

    To know what assert this is we need to check for the total combination of:
    - Test message
    - Test instance path
    - Expected value
    - Actual value
    Theoretically we can have a situation where a test has three different asserts, each and one with the same test
    message/test instance path/actual value/expected value but called within the same or different cycles. In order for
    us to handle all situations we need a simple algorithm that works according to:
    - Keep track of how many instances the combination of test message/test instance path/expected value/actual value
      we have. So for example, if we have called Assert(Exp := 5, Act := 5, 'Hello there', 'PRG.InstanceTestSuite.Test')
      two times in one cycle, we have two instances of that combination. This is done according to:
    - Iterate all existing reports.
      - If we have a new PLC-cycle, set the current detection-count to zero.
      - If new report does not match in any of the above fields, create it (together with current PLC-cycle).
        Also store the information that we have one instance of this combination and +1 on the detection-count.
      - If new report matches in all of the above, +1 in the detection-count. If this detection-count is larger than
        the stored detection-count for this combination, create a new report and add +1 to the storage of
        the detection-count.
*)
METHOD PUBLIC ReportResult
VAR_INPUT
    Expected : ANY;
    Actual : ANY;
    Message : Tc2_System.T_MaxString;
    TestInstancePath : Tc2_System.T_MaxString;
END_VAR
VAR_OUTPUT
    AlreadyReported : BOOL := FALSE;
END_VAR
VAR
    LocationIndex : UINT;
    DataTypesNotEquals : BOOL;
    DataSizeNotEquals : BOOL;
    DataContentNotEquals : BOOL;
    CurrentCycleCount : UDINT;
    IteratorCounter : UINT;
    DetectionCountTemp : UINT := 0;
    FoundOne : BOOL;
    AdditionalIdenticalAssert : BOOL;
END_VAR
IF NOT FirstCycleExecuted THEN
    GetCurrentTaskIndex();
    FirstCycleExecuted := TRUE;
END_IF

CurrentCycleCount := TwinCAT_SystemInfoVarList._TaskInfo[GetCurrentTaskIndex.index].CycleCount;
(* Is current cycle the same as the last call to this method?
   If not, reset the detection count *)
IF CurrentCycleCount <> CycleCount THEN
    CopyDetectionCountAndResetDetectionCountInThisCycle();
END_IF

FOR IteratorCounter := 1 TO TotalAsserts BY 1 DO
    IF F_IsAnyEqualToUnionValue(uExpectedOrActual := AssertResultInstances[IteratorCounter].AssertResult.Expected,
                                ExpectedOrActual := Expected) AND
       F_IsAnyEqualToUnionValue(uExpectedOrActual := AssertResultInstances[IteratorCounter].AssertResult.Actual,
                                ExpectedOrActual := Actual) AND
        AssertResultInstances[IteratorCounter].AssertResult.Message = Message AND
        AssertResultInstances[IteratorCounter].AssertResult.TestInstancePath = TestInstancePath THEN
        AssertResultInstances[IteratorCounter].DetectionCountThisCycle :=
            AssertResultInstances[IteratorCounter].DetectionCountThisCycle + 1;
            FoundOne := TRUE;
        IF AssertResultInstances[IteratorCounter].DetectionCountThisCycle >
                AssertResultInstances[IteratorCounter].DetectionCount THEN // This assert is new
                AdditionalIdenticalAssert := TRUE;
        END_IF
        EXIT;
    END_IF
END_FOR

(* If not found anything, create the first *)
IF NOT FoundOne THEN
    (* No existing match found, create a new entry *)
    AddAssertResult(Expected, Actual, Message, TestInstancePath);
    CreateAssertResultInstance(Expected := Expected, Actual := Actual, 
                               Message := Message, TestInstancePath := TestInstancePath);
(* An additional instance of this assert needs to be created *)
ELSIF AdditionalIdenticalAssert THEN
    AddAssertResult(Expected, Actual, Message, TestInstancePath);
(* In all other cases, this assert has already been reported, we don't need to do anything *)
ELSE
    AlreadyReported := TRUE;
END_IF

(* Update the cycle count *)
CycleCount := TwinCAT_SystemInfoVarList._TaskInfo[GetCurrentTaskIndex.index].CycleCount;
END_METHOD

END_FUNCTION_BLOCK

// POUs/FB_FileControl
{attribute 'hide_all_locals'}
FUNCTION_BLOCK FB_FileControl
VAR
    FileAccessMode : SysFile.ACCESS_MODE := SysFile.AM_WRITE_PLUS;
    FileHandle : SysFile.SysTypes.RTS_IEC_HANDLE;
END_VAR

// Closes the current file
METHOD PUBLIC Close : SysFile.SysTypes.RTS_IEC_RESULT;
IF FileHandle <> SysFile.SysTypes.RTS_INVALID_HANDLE THEN
    Close := SysFile.SysFileClose(hFile := FileHandle);
END_IF
END_METHOD

// Opens a file
METHOD PUBLIC Open : SysFile.SysTypes.RTS_IEC_RESULT;
VAR_INPUT
    FileName : Tc2_System.T_MaxString := 'filepath/output.xml'; // File name can contain an absolute or relative path to the file. Path entries must be separated with a Slash (/)
    FileAccessMode : SysFile.ACCESS_MODE := SysFile.ACCESS_MODE.AM_APPEND_PLUS;
END_VAR
FileHandle := SysFile.SysFileOpen(szFile := Filename,
                                  am := FileAccessMode,
                                  pResult := ADR(Open));
END_METHOD

METHOD Read : SysFile.SysTypes.RTS_IEC_RESULT;
VAR_INPUT
    pString : POINTER TO BYTE; // Call with ADR();
    Size : UDINT; // Call with SIZEOF(); 
END_VAR
VAR_OUTPUT
    FileSize : SysFile.SysTypes.RTS_IEC_SIZE;
END_VAR
IF FileHandle <> SysFile.SysTypes.RTS_INVALID_HANDLE THEN
    FileSize := SysFile.SysFileread(hFile := FileHandle, 
                                    pbyBuffer := pString,
                                    ulSize := Size,
                                    pResult := ADR(Read));
END_IF
END_METHOD

// Saves the contents of the buffer into a file
// Be sure to call Open() before calling Save()
METHOD Save : SysFile.SysTypes.RTS_IEC_RESULT;
VAR_INPUT
    pString : POINTER TO BYTE; // Call with ADR();
    Size : UDINT; // Call with SIZEOF();
END_VAR
IF FileHandle <> SysFile.SysTypes.RTS_INVALID_HANDLE THEN
    SysFile.SysFileWrite(hFile := FileHandle,
                         pbyBuffer := pString,
                         ulSize := Size,
                         pResult := ADR(Save));
END_IF
END_METHOD

END_FUNCTION_BLOCK

// POUs/FB_StringBuffer
(*
    This functionblock acts as an IO stream buffer for use with FB_XmlControl
*)
{attribute 'hide_all_locals'}
FUNCTION_BLOCK FB_StringBuffer 
VAR
    pString : POINTER TO BYTE;
    udiLength : UDINT;
    udiSizeOf : UDINT;
END_VAR

// Appends a string to the buffer
PROPERTY Append : Tc2_System.T_MaxString
SET
VAR
    pByteIn : POINTER TO BYTE;
    pByteBuffer : POINTER TO BYTE;
END_VAR
pByteIn := ADR(Append); 
pByteBuffer := pString + udiLength;
WHILE pByteIn^ <> 0 AND(udiLength < udiSizeOf ) DO
    pByteBuffer^ := pByteIn^;
    udiLength := udiLength + 1;
    pByteIn := pByteIn + 1;
    pByteBuffer := pByteBuffer + 1;
END_WHILE;

pByteBuffer := pString + udiLength; (* String End *)
pByteBuffer^ := 0;
END_SET
END_PROPERTY

// Read current Buffersize
PROPERTY BufferSize : UDINT
GET
BufferSize := udiSizeOf;
END_GET
END_PROPERTY

(*
    Copies a string from the character buffer
*)
METHOD Copy : Tc2_System.T_MaxString
VAR_INPUT
    udiStart : UDINT;
    udiEnd : UDINT;
END_VAR
VAR_OUTPUT
    udiCopyLen : UDINT;
    XmlError : E_XmlError;
END_VAR
VAR
    udiLoop : UDINT;
    pByteCopy : POINTER TO BYTE;
    pByteBuffer : POINTER TO BYTE;
END_VAR
udiLoop := 0;
pByteCopy := ADR(Copy);
pByteBuffer := pString + udiStart - 1;

WHILE(udiLoop < SIZEOF(Copy)) AND udiStart - 1 + udiLoop < udiLength AND udiStart + udiLoop < udiEnd DO
    pByteCopy^ := pByteBuffer^;
    udiLoop := udiLoop + 1;
    pByteCopy := ADR(Copy) + udiLoop;
    pByteBuffer := pString + udiStart + udiLoop -1;
END_WHILE;

IF udiLoop = SIZEOF(Copy) THEN
    XmlError := E_XmlError.ErrorStringLen;
ELSIF udiStart - 1 + udiLoop = udiLength THEN
    XmlError := E_XmlError.ErrorMaxBufferLen;
ELSE
    XmlError := E_XmlError.OK;
END_IF;

pByteCopy^ := 0;
udiCopyLen :=  udiLoop;
END_METHOD

METHOD CutOff : STRING
VAR_INPUT
    udiStartPos : UDINT;
END_VAR
VAR_OUTPUT
    udiCutLen : UDINT; 
    XmlError : E_XmlError;
END_VAR
VAR
    iLoop : UDINT;
    pByteCut : POINTER TO BYTE;
    pByteBuffer : POINTER TO BYTE;
END_VAR
iLoop := 0;
pByteCut := ADR(CutOff);
pByteBuffer := pString + udiStartPos - 1;

WHILE pByteBuffer^ <> 0 AND(iLoop < SIZEOF(CutOff)) AND udiStartPos -1  + iLoop < udiLength DO
    pByteCut^ := pByteBuffer^;
    iLoop := iLoop + 1;
    pByteCut := ADR(CutOff) + iLoop;
    pByteBuffer := pString + udiStartPos - 1 + iLoop;
END_WHILE;

IF pByteBuffer^ = 0 THEN
    XmlError := E_XmlError.OK;
ELSIF iLoop = SIZEOF(CutOff) THEN
    XmlError := E_XmlError.ErrorStringLen;
ELSIF udiStartPos -1 + iLoop = udiLength THEN
    XmlError := E_XmlError.ErrorMaxBufferLen;
END_IF;

pByteCut^ := 0;
udiLength := udiStartPos -1;

pByteBuffer := pString + udiStartPos - 1;
pByteBuffer^ := 0;

udiCutLen := iLoop;
END_METHOD

(* 
    Find a searchstring in the buffer and returns its position.
    It's possible to add a preffered startposition within buffer
*)
METHOD Find : UDINT
VAR_INPUT
    sSearchString : STRING;
    udiStartPos : UDINT;
END_VAR
VAR
    udiLoop : UDINT;
    iSearch : UDINT;
    pBuffer : POINTER TO BYTE;
    pSearch : POINTER TO BYTE;
END_VAR
udiLoop := 0;
iSearch := 0;

pBuffer := pString + udiStartPos;
pSearch := ADR( sSearchString);

WHILE(pSearch^ <> 0 ) AND udiLoop + udiStartPos < udiLength DO
    IF pBuffer^ <> pSearch^ THEN
        udiLoop := udiLoop + 1;
        pBuffer := pString + udiStartPos + udiLoop;
        pSearch := ADR( sSearchString);
        iSearch := 0;
    ELSE
        iSearch := iSearch +1;
        pBuffer := pString + udiStartPos + udiLoop + iSearch;
        pSearch := ADR( sSearchString ) + iSearch;
    END_IF;
END_WHILE;
Find := udiLoop + 1 + udiStartPos;
END_METHOD

METHOD FindBack : UDINT
VAR_INPUT
    sSearchString : Tc2_System.T_MaxString;
END_VAR
VAR
    udiLoop : UDINT;
    udiSearch : UDINT;
    pBuffer : POINTER TO BYTE;
    pSearch : POINTER TO BYTE;
END_VAR
udiLoop := 0;
udiSearch := 0;

pBuffer := pString + udiLength;
pSearch := ADR( sSearchString);

WHILE(pSearch^ <> 0 ) AND udiLoop < udiLength DO
    IF pBuffer^ <> pSearch^ THEN
        udiLoop := udiLoop + 1;
        pBuffer := pString + udiLength - udiLoop;
        pSearch := ADR( sSearchString);
        udiSearch := 0;
    ELSE
        udiSearch := udiSearch +1;
        pBuffer := pString + udiLength - udiLoop + udiSearch;
        pSearch := ADR( sSearchString ) + udiSearch;
    END_IF;
END_WHILE;
FindBack :=  udiLength - udiLoop + 1;
END_METHOD

PROPERTY Length : UDINT
GET
Length := udiLength;
END_GET
SET
udiLength := Length;
END_SET
END_PROPERTY

(* Sets the Buffer *)
METHOD Set : BOOL;
VAR_INPUT
    // Set buffer adress (ADR ...)
    pbyAdr : POINTER TO BYTE;
    // Set buffer size (SIZEOF ...)
    udiSize : UDINT;
END_VAR
IF (pbyAdr = 0)OR (udiSize = 0) THEN
    Set := FALSE;
    RETURN;
END_IF;

udiSizeOf := udiSize;
pString := pbyAdr;

Set := TRUE;
END_METHOD

END_FUNCTION_BLOCK

// POUs/FB_XmlControl
(*
Organizes parsing and composing of XML data. Data can be treated as STRING or char array.
Filebuffersize is default 4096 bytes and can be set via Gvl_Param_XmlControl

Usage example:

1. Initiate
    VAR
        XML : XML_Control;
        Buffer: STRING(GVL_Param_XmlControl.udiMaxFileSize);
        //or
        Buffer: ARRAY [0..GVL_Param_XmlControl.udiMaxFileSize] OF CHAR;
    END_VAR

    XML.pBuffer: = ADR (buffer);
    XML.LenBuffer: = SIZEOF (buffer);


    Add your own preferred fileheader like:
    XML: <?xml version=\"1.0\" encoding=\"UTF-8\"?>

    XML.WriteDocumentHeader( '<?xml version=\"1.0\" encoding=\"UTF-8\"?>');

2. Compose a tag with a parameters:
XML: <MyTag ParaName = "11" />

    XML.newTag(sTagName: = 'MyTag');
    XML.newPara(sName: = 'ParaName', sPara: = sValue);
    XML.CloseTag();


3. Add tag value:
XML: <MyTag> MyText </ MyTag>

    XML.newTag(sName := 'MyTag');
    XML.newTagData(sTagData :='MyText');
    XML.CloseTag();


4. Jump to the beginning of the XML data
XML.toStartBuffer();


5. Add a comment:
XML: <!-- MyComment -->

    XML.newComment(sTagName: = 'MyComment');

6. Returns the next tag from the current position in buffer
XML.NextTag();


7. Output the parameter of the tag
XML.NextPara(sPara: = LastValue);
Feedback: sPara returns the value found (string)

*)
{attribute 'hide_all_locals'}
FUNCTION_BLOCK FB_XmlControl
VAR
    Buffer : FB_StringBuffer;
    TagList : FB_StringBuffer;
    sTags : Tc2_System.T_MaxString;
    TagListSeek : FB_StringBuffer;
    sTagsSeek : STRING;
    Tag : FB_StringBuffer;
    sTag : Tc2_System.T_MaxString;
    xTagOpen: BOOL;
    iSelect : UDINT;
    iSelectStart : UDINT;
    iSelectEnd : UDINT;
    iSelectStartPara : UDINT;
    iSelectEndPara : UDINT;
    iSelectTagClose : UDINT;
    iSelectStartValue : UDINT;
    iSelectEndValue : UDINT;
    udiSearchPos : UDINT; 
END_VAR
VAR CONSTANT
    TAG_OPEN : STRING(1) := '<';
    TAG_CLOSE : STRING(1) := '>';
    END_TAG_CLOSE : STRING(4) := '/>$R$L';
    SPACE : STRING(1) := ' ';
    EQUALS : STRING(1) := '=';
    QUOTE : STRING(1) := '"';
    BACK_SLASH : STRING(1) := '\';
    FORWARD_SLASH : STRING(1) := '/';
    OPEN_COMMENT : STRING(5) := '<!-- ';
    CLOSE_COMMENT : STRING(4) := ' -->';
END_VAR

(* 
    Clears the contents of the entire buffer
*)
METHOD PUBLIC ClearBuffer
udiSearchPos := 0;
TagListSeek.Length := 0;
Buffer.Length := 0;
sTagsSeek := '';
sTag := '';
END_METHOD

(*
    Closes a Tag:
    XML: <MyTag />

    Method: XML.CloseTag();
*)
METHOD PUBLIC CloseTag : Tc2_System.T_MaxString
IF xTagOpen THEN
    Buffer.Append := END_TAG_CLOSE;
    iSelect := TagList.FindBack(sSearchString := FORWARD_SLASH);
    CloseTag := TagList.CutOff(udiStartPos:= iSelect);
    xTagOpen := FALSE;
ELSE
    iSelect := TagList.FindBack(sSearchString := FORWARD_SLASH);
    CloseTag := TagList.CutOff(udiStartPos:= iSelect);
    Buffer.Append := TAG_OPEN;
    Buffer.Append := CloseTag;
    Buffer.Append := TAG_CLOSE;
END_IF
END_METHOD

PROPERTY Length : UDINT
GET
Length := Buffer.Length;
END_GET
END_PROPERTY

(*
    Adds a comment;
    XML: <!-- MyComment -->

    XML.NewComment(Comment: = 'MyComment');
*)
METHOD PUBLIC NewComment
VAR_INPUT
    Comment : Tc2_System.T_MaxString;
END_VAR
IF xTagOpen THEN
    Buffer.Append := TAG_CLOSE;
    xTagOpen := FALSE;
END_IF;
Buffer.Append := OPEN_COMMENT;
Buffer.Append := Comment;
Buffer.Append := CLOSE_COMMENT;
END_METHOD

(*
    Must be called after opening a new tag

    XML.NewParameter(Name: = 'ParaName', Value: = 'Value');
*)
METHOD PUBLIC NewParameter
VAR_INPUT
    Name : Tc2_System.T_MaxString;
    Value : Tc2_System.T_MaxString;
END_VAR
Buffer.Append := SPACE;  
Buffer.Append := Name;
Buffer.Append := EQUALS; 
Buffer.Append := QUOTE; 
Buffer.Append := Value;
Buffer.Append := QUOTE;
END_METHOD

(*
    Creates a new Tag:
    XML: <MyTag>

    XML.NewTag(Name: = 'MyTag');
*)
METHOD PUBLIC NewTag
VAR_INPUT
    Name : Tc2_System.T_MaxString;
END_VAR
IF xTagOpen THEN
    Buffer.Append := TAG_CLOSE;
END_IF;
Buffer.Append := TAG_OPEN;
Buffer.Append := Name;
xTagOpen := TRUE;
TagList.Append := FORWARD_SLASH;
TagList.Append := Name;
END_METHOD

METHOD PUBLIC NewTagData
VAR_INPUT
    Data : Tc2_System.T_MaxString;
END_VAR
Buffer.Append := TAG_CLOSE;
Buffer.Append := Data;
xTagOpen := FALSE;
END_METHOD

METHOD PUBLIC NextParameter : Tc2_System.T_MaxString;
VAR_OUTPUT
    Parameter : Tc2_System.T_MaxString;
END_VAR
VAR
    Name : Tc2_System.T_MaxString;
END_VAR
iSelectEndPara := Buffer.Find(sSearchString := EQUALS, udiStartPos := iSelectStartPara);
IF iSelectStartPara < iSelectEnd AND iSelectEndPara < iSelectEnd THEN
    Name := Buffer.Copy( udiStart := iSelectStartPara + 1, udiEnd := iSelectEndPara);
    iSelectStartValue := Buffer.Find(sSearchString := QUOTE, udiStartPos := iSelectEndPara);
    iSelectEndValue := Buffer.Find(sSearchString := QUOTE, udiStartPos := iSelectStartValue);
    Parameter := Buffer.Copy( udiStart := iSelectStartValue + 1, udiEnd := iSelectEndValue);
    iSelectStartPara := iSelectEndValue + 1;
ELSE
    iSelectEndValue := Buffer.Find(sSearchString := TAG_OPEN, udiStartPos := udiSearchPos);
    Name := Buffer.Copy( udiStart := udiSearchPos + 1, udiEnd := iSelectEndValue); 
END_IF;
NextParameter := Name;
END_METHOD

METHOD PUBLIC NextTag : Tc2_System.T_MaxString
iSelectStart := Buffer.Find(sSearchString := TAG_OPEN, udiStartPos := udiSearchPos);
iSelectEnd := Buffer.Find(sSearchString := TAG_CLOSE, udiStartPos := iSelectStart);
iSelectStartPara := Buffer.Find(sSearchString := SPACE, udiStartPos := iSelectStart);
iSelectTagClose := Buffer.Find(sSearchString := FORWARD_SLASH, udiStartPos := iSelectStart);
IF iSelectStart < Buffer.Length AND iSelectEnd < Buffer.Length THEN
    udiSearchPos := iSelectEnd;
    sTag := Buffer.Copy( udiStart:= iSelectStart + 1, udiEnd:= iSelectEnd);
    IF iSelectEnd < iSelectStartPara THEN
        NextTag := Buffer.Copy( udiStart:= iSelectStart + 1, udiEnd:= iSelectEnd);
    ELSE
        NextTag := Buffer.Copy( udiStart:= iSelectStart + 1, udiEnd:= iSelectStartPara);
    END_IF;
    IF iSelectTagClose = iSelectStart +1 THEN
        iSelect := TagListSeek.FindBack(sSearchString := FORWARD_SLASH);
        TagListSeek.CutOff(udiStartPos:= iSelect);
    ELSIF iSelectTagClose > iSelectStart AND iSelectTagClose < iSelectEnd THEN
        TagListSeek.Append := '/';
        TagListSeek.Append := NextTag;
        iSelect := TagListSeek.FindBack(sSearchString := FORWARD_SLASH);
        TagListSeek.CutOff(udiStartPos:= iSelect);
    ELSE
        TagListSeek.Append := FORWARD_SLASH;
        TagListSeek.Append := NextTag;
    END_IF;
ELSE
    udiSearchPos := Buffer.Length;
    NextTag := '';
END_IF;
END_METHOD

METHOD PUBLIC SetBuffer
VAR_INPUT
    pString : POINTER TO BYTE;
    iSizeOf : UDINT;
END_VAR
Buffer.Set(pbyAdr := pString, udiSize := iSizeOf);
TagList.Set(pbyAdr := ADR(sTags), udiSize := SIZEOF(sTags));
TagListSeek.Set(pbyAdr := ADR(sTagsSeek), udiSize := SIZEOF(sTagsSeek));
Tag.Set(pbyAdr := ADR(sTag), udiSize := SIZEOF(sTag));
END_METHOD

(*
    Jump to the beginning of the XML data
    XML.ToStartBuffer();
*)
METHOD PUBLIC ToStartBuffer
udiSearchPos := 0;
TagListSeek.Length := 0;
sTagsSeek := '';
sTag := '';
END_METHOD

(*
    Add your own preffered fileheader like:
    XML: <?xml version=\"1.0\" encoding=\"UTF-8\"?>

    XML.WriteDocumentHeader('<?xml version=\"1.0\" encoding=\"UTF-8\"?>');

*)
METHOD PUBLIC WriteDocumentHeader
VAR_INPUT
    Header : Tc2_System.T_MaxString;
END_VAR
Buffer.Append := Header;
END_METHOD

END_FUNCTION_BLOCK

// POUs/FB_TcUnitRunner
(*
    This function block is responsible for holding track of the tests and executing them.
*)
FUNCTION_BLOCK FB_TcUnitRunner
VAR
    (* Indication of whether all test suites have reported that they are finished *)
    AllTestSuitesFinished : BOOL := FALSE;

    (* Prints the results to ADS so that Visual Studio can display the results.
       This test result formatter can be replaced with something else than ADS *)
    ADSTestResultFormatter : FB_ADSTestResultFormatter;
    TestResultPrinter : I_TestResultFormatter := ADSTestResultFormatter;

    (* These variables (statistics) are occupied once all tests are complete *)
    NumberOfTestSuitesFinished : UINT := 0;
    NumberOfTestCases : UINT := 0;
    NumberOfFailedTestCases : UINT := 0;
    NumberOfSuccessfulTestCases : UINT := 0;

    (* Indication of that the printing of test results is complete *)
    DonePrintingTestResults : BOOL;

    (* If this flag is set, it means that some external event triggered the
       request to abort running the test suites *)
    AbortRunningTestSuites : BOOL;
END_VAR

(* This function sets a flag which makes the runner stop running the tests
   in the test suites *)
METHOD PUBLIC AbortRunningTestSuiteTests
AbortRunningTestSuites := TRUE;
END_METHOD

METHOD RunTestSuiteTests
VAR
    Counter : UINT := 0;
    BusyPrinting : BOOL;

    (* We need to hold a temporary state of the statistics (failed, successful, total number of test cases etc)
       as we don't consider the tests to be completely finished until all test suites have executed completely.
       The reason we want to do it this way is because a test suite can run over several cycles. Only once all tests
       are finished (which might take many cycles), do we gather correct statistics *)
    NumberOfTestSuitesFinished_Temp : UINT := 0;
    NumberOfTestCases_Temp : UINT := 0;
    NumberOfFailedTestCases_Temp : UINT := 0;
    NumberOfSuccessfulTestCases_Temp : UINT := 0;
END_VAR
IF NOT AllTestSuitesFinished THEN
    IF GVL_TcUnit.NumberOfInitializedTestSuites = 0 THEN
        AllTestSuitesFinished := TRUE;
    ELSIF GVL_TcUnit.NumberOfInitializedTestSuites > 0 THEN
        FOR Counter := 1 TO GVL_TcUnit.NumberOfInitializedTestSuites BY 1 DO
            IF GVL_TcUnit.TestSuiteAddresses[Counter]^.AreAllTestsFinished() THEN
                NumberOfTestSuitesFinished_Temp := NumberOfTestSuitesFinished_Temp + 1;
                NumberOfTestCases_Temp := GVL_TcUnit.TestSuiteAddresses[Counter]^.GetNumberOfTests() + NumberOfTestCases_Temp;
                NumberOfFailedTestCases_Temp := GVL_TcUnit.TestSuiteAddresses[Counter]^.GetNumberOfFailedTests() + NumberOfFailedTestCases_Temp;
                NumberOfSuccessfulTestCases_Temp := GVL_TcUnit.TestSuiteAddresses[Counter]^.GetNumberOfSuccessfulTests() + NumberOfSuccessfulTestCases_Temp;
            ELSE
                GVL_TcUnit.CurrentTestSuiteBeingCalled := GVL_TcUnit.TestSuiteAddresses[Counter];
                GVL_TcUnit.CurrentTestSuiteBeingCalled^();
            END_IF
        END_FOR
        (* Check if some event triggered an abortion of running the tests, in that case abort it now.
           This can be accomplished by setting the result of the test suites run to finished. *)
        IF AbortRunningTestSuites THEN
            NumberOfTestSuitesFinished_Temp := GVL_TcUnit.NumberOfInitializedTestSuites;
		END_IF
        IF NumberOfTestSuitesFinished_Temp = GVL_TcUnit.NumberOfInitializedTestSuites THEN
            (* Copy the final results over *)
            NumberOfTestSuitesFinished := NumberOfTestSuitesFinished_Temp;
            NumberOfTestCases := NumberOfTestCases_Temp;
            NumberOfFailedTestCases := NumberOfFailedTestCases_Temp;
            NumberOfSuccessfulTestCases := NumberOfSuccessfulTestCases_Temp;
            AllTestSuitesFinished := TRUE;
        END_IF
    END_IF
END_IF

IF AllTestSuitesFinished THEN
    IF NOT DonePrintingTestResults THEN
        TestResultPrinter.Format(NumberOfTestSuites := NumberOfTestSuitesFinished,
                                 NumberOfTestCases := NumberOfTestCases,
                                 NumberOfSuccessfulTestCases := NumberOfSuccessfulTestCases,
                                 NumberOfFailedTestCases := NumberOfFailedTestCases,
                                 Busy => BusyPrinting);
        DonePrintingTestResults := NOT BusyPrinting;
    END_IF
END_IF

(* Run the buffered ADS logger *)
GVL_TcUnit.AdsLogger();
END_METHOD

END_FUNCTION_BLOCK

// POUs/FB_TestSuite
(* This function block is responsible for holding the internal state of the test suite.
   Every test suite can have one or more tests, and every test can do one or more asserts.
   It's also responsible for providing all the assert-methods for asserting different data types.
   Only failed assertions are recorded.
*)
{attribute 'call_after_init'}
{attribute 'reflection'}
FUNCTION_BLOCK FB_TestSuite
VAR
    {attribute 'instance-path'}
    {attribute 'noinit'}
    InstancePath : Tc2_System.T_MaxString;

    (* We need to have access to specific information of the current task that this test suite
       is executed in. This is for instance necessary when we need to know whether a test is
       defined already. The definition of a test that is defined already is that we call on it
       with the same name twice in the same cycle *)
    GetCurrentTaskIndex : Tc2_System.GETCURTASKINDEX;

    NumberOfTests : UINT := 0;
    Tests : ARRAY[1..GVL_Param_TcUnit.MaxNumberOfTestsForEachTestSuite] OF FB_Test;
    (* Rising trigger of whether we have already notified the user of that the test name pointed to by the current
       position is a duplicate *)
    TestDuplicateNameTrigger : ARRAY[1..GVL_Param_TcUnit.MaxNumberOfTestsForEachTestSuite] OF Tc2_Standard.R_TRIG;
    (* Last cycle count index for a specific test. Used to detect whether this test has already been defined in the
       current test suite *)
    TestCycleCountIndex : ARRAY[1..GVL_Param_TcUnit.MaxNumberOfTestsForEachTestSuite] OF UDINT;

    AssertResults : FB_AssertResultStatic;
    AssertArrayResult : FB_AssertArrayResultStatic;

    (* Prints the failed asserts to ADS so that Visual Studio can display the assert message.
       This assert formatter can be replaced with something else than ADS *)
    ADSAssertMessageFormatter : FB_ADSAssertMessageFormatter;
    AssertMessageFormatter : I_AssertMessageFormatter := ADSAssertMessageFormatter;
END_VAR

METHOD PUBLIC AddTest
VAR_INPUT
    TestName : Tc2_System.T_MaxString;
END_VAR
VAR
    IteratorCounter : UINT;
    ErrorMessage : Tc2_System.T_MaxString;
    TestInstancePath : Tc2_System.T_MaxString;
    FunctionCallResult : DINT;
    CycleCount : UDINT;
    TestWithThisNameAlreadyExists : BOOL := FALSE;
    LowerCasedTestName : Tc2_System.T_MaxString;
    TrimmedTestName : Tc2_System.T_MaxString;
END_VAR
GVL_TcUnit.IgnoreCurrentTest := FALSE; // Reset the ignore current test flag

TrimmedTestName := Tc2_Utilities.F_LTrim(in := TestName);
TrimmedTestName := Tc2_Utilities.F_RTrim(in := TrimmedTestName);
LowerCasedTestName := Tc2_Utilities.F_ToLCase(in := TrimmedTestName);

(* Check if this test should be disabled *)
IF Tc2_Utilities.FIND(STR1 := LowerCasedTestName, STR2 := 'disabled_') = 1 THEN
    GVL_TcUnit.IgnoreCurrentTest := TRUE;
    RETURN;
END_IF

GetCurrentTaskIndex(); // Gets the task index of where this function block instance is being run in

(* Check if the test name already exists. Make sure there are no other tests with the same name already
   added for this test suite *)

CycleCount := TwinCAT_SystemInfoVarList._TaskInfo[GetCurrentTaskIndex.index].CycleCount;

(* Iterate all the test names that up to this point have been added for this test suite *)
FOR IteratorCounter := 1 TO NumberOfTests BY 1 DO
    IF Tests[IteratorCounter].GetName() = TrimmedTestName THEN
        TestWithThisNameAlreadyExists := TRUE;
        (* Check if a test with this name has already been called in this PLC cycle *)
        IF TestCycleCountIndex[IteratorCounter] = CycleCount THEN
            GVL_TcUnit.IgnoreCurrentTest := TRUE;
            (* A test with this name already exists for this test suite and has already been called in this cycle.
               Send a message notification, but only if we have not done so already. *)
            TestDuplicateNameTrigger[IteratorCounter](CLK := TRUE);
            IF TestDuplicateNameTrigger[IteratorCounter].Q THEN // Rising edge detected. We have not reported this before
                TestInstancePath := F_RemoveInstancePathAndProjectNameFromTestInstancePath(TestInstancePath :=
                                                                                           GVL_TcUnit.CurrentTestSuiteBeingCalled^.GetInstancePath());
                ErrorMessage := 'Test with name $'%s$' already exists in test suite $'';
                ErrorMessage := Tc2_Standard.CONCAT(STR1 := ErrorMessage, STR2 := TestInstancePath);
                ErrorMessage := Tc2_Standard.CONCAT(STR1 := ErrorMessage, STR2 := '$'');
                GVL_TcUnit.AdsLogger.WriteLog(MsgFmtStr := ErrorMessage,
                                              StrArg := TrimmedTestName);
            END_IF
        END_IF
        TestCycleCountIndex[IteratorCounter] := CycleCount;
    END_IF
END_FOR

IF NOT TestWithThisNameAlreadyExists THEN
    (* Test has not been found. Add it. *)
    Tests[IteratorCounter].SetName(Name := TrimmedTestName);
    NumberOfTests := NumberOfTests + 1;
    TestCycleCountIndex[NumberOfTests] := CycleCount;
END_IF
END_METHOD

METHOD PRIVATE AddTestNameToInstancePath : Tc2_System.T_MaxString
VAR_INPUT
    TestInstancePath : Tc2_System.T_MaxString;
END_VAR
VAR
    CompleteTestInstancePath : Tc2_System.T_MaxString;
END_VAR
CompleteTestInstancePath := Tc2_Utilities.CONCAT(STR1 := TestInstancePath, STR2 := '@');
AddTestNameToInstancePath := Tc2_Utilities.CONCAT(STR1 := CompleteTestInstancePath, STR2 := GVL_TcUnit.CurrentTestNameBeingCalled);
END_METHOD

METHOD PUBLIC AreAllTestsFinished : BOOL
VAR
    Counter : UINT;

    GetCurTaskIndex : Tc2_System.GETCURTASKINDEX;
END_VAR
AreAllTestsFinished := FALSE;

IF NumberOfTests > 0 THEN
    AreAllTestsFinished := TRUE;
    FOR Counter := 1 TO GetNumberOfTests() BY 1 DO
        AreAllTestsFinished := AreAllTestsFinished AND Tests[Counter].IsFinished();
    END_FOR
END_IF

(* If we have been running at least one cycle and no tests are registered it means that this testsuite is empty
   and doesn't contain any test cases. In that case, add a warning message and ignore this testsuite. *)
GetCurTaskIndex();
IF NumberOfTests = 0 AND NOT TwinCAT_SystemInfoVarList._TaskInfo[GetCurTaskIndex.index].FirstCycle THEN
    AreAllTestsFinished := TRUE;
END_IF
END_METHOD

